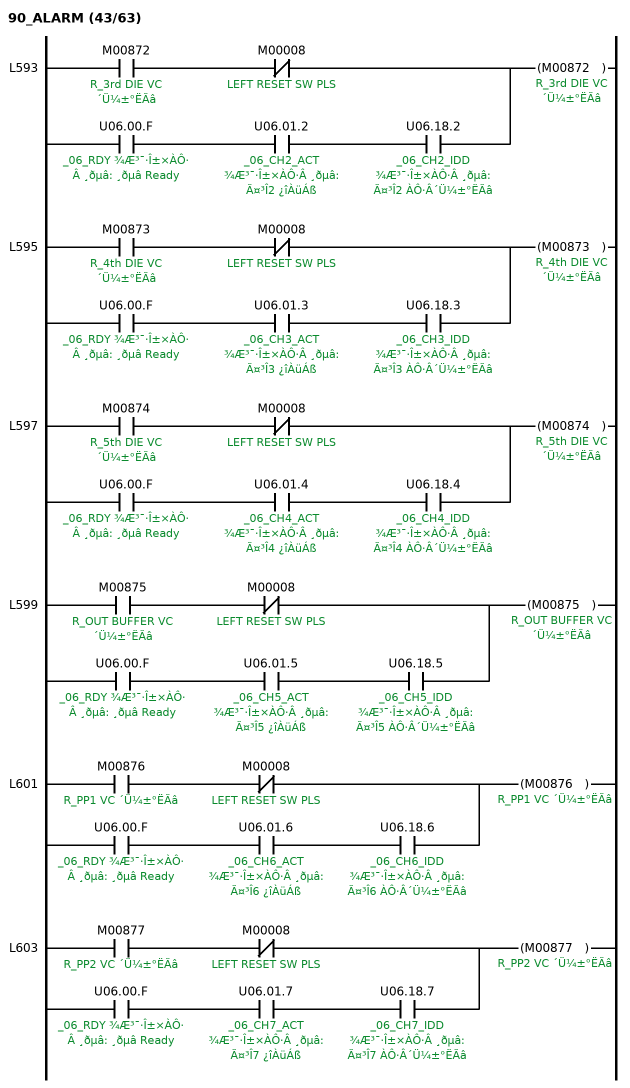
[picture p408: 90_ALARM rungs L593-L603]
; L593
LOAD      M00872	// R_3rd DIE VC ´Ü¼±°ËÃâ
AND NOT   M00008	// LEFT RESET SW PLS
LOAD      U06.00.F	// _06_RDY ¾Æ³¯·Î±×ÀÔ·Â ¸ðµâ: ¸ðµâ Ready
AND       U06.01.2	// _06_CH2_ACT ¾Æ³¯·Î±×ÀÔ·Â ¸ðµâ: Ã¤³Î2 ¿îÀüÁß
AND       U06.18.2	// _06_CH2_IDD ¾Æ³¯·Î±×ÀÔ·Â ¸ðµâ: Ã¤³Î2 ÀÔ·Â´Ü¼±°ËÃâ
OR LOAD
OUT       M00872	// R_3rd DIE VC ´Ü¼±°ËÃâ
; L595
LOAD      M00873	// R_4th DIE VC ´Ü¼±°ËÃâ
AND NOT   M00008	// LEFT RESET SW PLS
LOAD      U06.00.F	// _06_RDY ¾Æ³¯·Î±×ÀÔ·Â ¸ðµâ: ¸ðµâ Ready
AND       U06.01.3	// _06_CH3_ACT ¾Æ³¯·Î±×ÀÔ·Â ¸ðµâ: Ã¤³Î3 ¿îÀüÁß
AND       U06.18.3	// _06_CH3_IDD ¾Æ³¯·Î±×ÀÔ·Â ¸ðµâ: Ã¤³Î3 ÀÔ·Â´Ü¼±°ËÃâ
OR LOAD
OUT       M00873	// R_4th DIE VC ´Ü¼±°ËÃâ
; L597
LOAD      M00874	// R_5th DIE VC ´Ü¼±°ËÃâ
AND NOT   M00008	// LEFT RESET SW PLS
LOAD      U06.00.F	// _06_RDY ¾Æ³¯·Î±×ÀÔ·Â ¸ðµâ: ¸ðµâ Ready
AND       U06.01.4	// _06_CH4_ACT ¾Æ³¯·Î±×ÀÔ·Â ¸ðµâ: Ã¤³Î4 ¿îÀüÁß
AND       U06.18.4	// _06_CH4_IDD ¾Æ³¯·Î±×ÀÔ·Â ¸ðµâ: Ã¤³Î4 ÀÔ·Â´Ü¼±°ËÃâ
OR LOAD
OUT       M00874	// R_5th DIE VC ´Ü¼±°ËÃâ
; L599
LOAD      M00875	// R_OUT BUFFER VC ´Ü¼±°ËÃâ
AND NOT   M00008	// LEFT RESET SW PLS
LOAD      U06.00.F	// _06_RDY ¾Æ³¯·Î±×ÀÔ·Â ¸ðµâ: ¸ðµâ Ready
AND       U06.01.5	// _06_CH5_ACT ¾Æ³¯·Î±×ÀÔ·Â ¸ðµâ: Ã¤³Î5 ¿îÀüÁß
AND       U06.18.5	// _06_CH5_IDD ¾Æ³¯·Î±×ÀÔ·Â ¸ðµâ: Ã¤³Î5 ÀÔ·Â´Ü¼±°ËÃâ
OR LOAD
OUT       M00875	// R_OUT BUFFER VC ´Ü¼±°ËÃâ
; L601
LOAD      M00876	// R_PP1 VC ´Ü¼±°ËÃâ
AND NOT   M00008	// LEFT RESET SW PLS
LOAD      U06.00.F	// _06_RDY ¾Æ³¯·Î±×ÀÔ·Â ¸ðµâ: ¸ðµâ Ready
AND       U06.01.6	// _06_CH6_ACT ¾Æ³¯·Î±×ÀÔ·Â ¸ðµâ: Ã¤³Î6 ¿îÀüÁß
AND       U06.18.6	// _06_CH6_IDD ¾Æ³¯·Î±×ÀÔ·Â ¸ðµâ: Ã¤³Î6 ÀÔ·Â´Ü¼±°ËÃâ
OR LOAD
OUT       M00876	// R_PP1 VC ´Ü¼±°ËÃâ
; L603
LOAD      M00877	// R_PP2 VC ´Ü¼±°ËÃâ
AND NOT   M00008	// LEFT RESET SW PLS
LOAD      U06.00.F	// _06_RDY ¾Æ³¯·Î±×ÀÔ·Â ¸ðµâ: ¸ðµâ Ready
AND       U06.01.7	// _06_CH7_ACT ¾Æ³¯·Î±×ÀÔ·Â ¸ðµâ: Ã¤³Î7 ¿îÀüÁß
AND       U06.18.7	// _06_CH7_IDD ¾Æ³¯·Î±×ÀÔ·Â ¸ðµâ: Ã¤³Î7 ÀÔ·Â´Ü¼±°ËÃâ
OR LOAD
OUT       M00877	// R_PP2 VC ´Ü¼±°ËÃâ

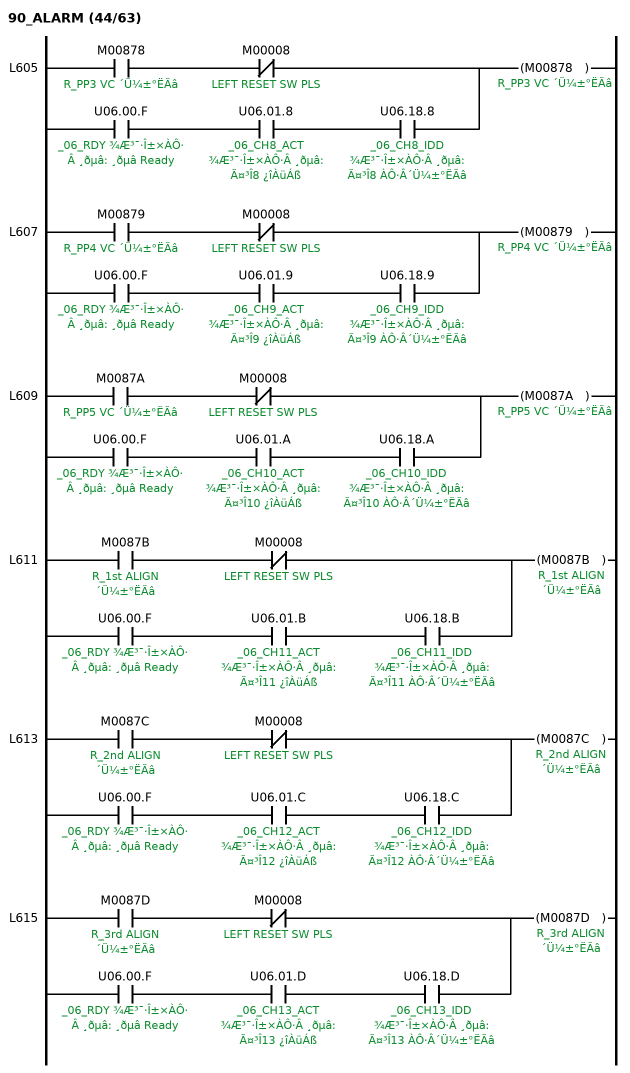
; L605
LOAD      M00878	// R_PP3 VC ´Ü¼±°ËÃâ
AND NOT   M00008	// LEFT RESET SW PLS
LOAD      U06.00.F	// _06_RDY ¾Æ³¯·Î±×ÀÔ·Â ¸ðµâ: ¸ðµâ Ready
AND       U06.01.8	// _06_CH8_ACT ¾Æ³¯·Î±×ÀÔ·Â ¸ðµâ: Ã¤³Î8 ¿îÀüÁß
AND       U06.18.8	// _06_CH8_IDD ¾Æ³¯·Î±×ÀÔ·Â ¸ðµâ: Ã¤³Î8 ÀÔ·Â´Ü¼±°ËÃâ
OR LOAD
OUT       M00878	// R_PP3 VC ´Ü¼±°ËÃâ
; L607
LOAD      M00879	// R_PP4 VC ´Ü¼±°ËÃâ
AND NOT   M00008	// LEFT RESET SW PLS
LOAD      U06.00.F	// _06_RDY ¾Æ³¯·Î±×ÀÔ·Â ¸ðµâ: ¸ðµâ Ready
AND       U06.01.9	// _06_CH9_ACT ¾Æ³¯·Î±×ÀÔ·Â ¸ðµâ: Ã¤³Î9 ¿îÀüÁß
AND       U06.18.9	// _06_CH9_IDD ¾Æ³¯·Î±×ÀÔ·Â ¸ðµâ: Ã¤³Î9 ÀÔ·Â´Ü¼±°ËÃâ
OR LOAD
OUT       M00879	// R_PP4 VC ´Ü¼±°ËÃâ
; L609
LOAD      M0087A	// R_PP5 VC ´Ü¼±°ËÃâ
AND NOT   M00008	// LEFT RESET SW PLS
LOAD      U06.00.F	// _06_RDY ¾Æ³¯·Î±×ÀÔ·Â ¸ðµâ: ¸ðµâ Ready
AND       U06.01.A	// _06_CH10_ACT ¾Æ³¯·Î±×ÀÔ·Â ¸ðµâ: Ã¤³Î10 ¿îÀüÁß
AND       U06.18.A	// _06_CH10_IDD ¾Æ³¯·Î±×ÀÔ·Â ¸ðµâ: Ã¤³Î10 ÀÔ·Â´Ü¼±°ËÃâ
OR LOAD
OUT       M0087A	// R_PP5 VC ´Ü¼±°ËÃâ
; L611
LOAD      M0087B	// R_1st ALIGN ´Ü¼±°ËÃâ
AND NOT   M00008	// LEFT RESET SW PLS
LOAD      U06.00.F	// _06_RDY ¾Æ³¯·Î±×ÀÔ·Â ¸ðµâ: ¸ðµâ Ready
AND       U06.01.B	// _06_CH11_ACT ¾Æ³¯·Î±×ÀÔ·Â ¸ðµâ: Ã¤³Î11 ¿îÀüÁß
AND       U06.18.B	// _06_CH11_IDD ¾Æ³¯·Î±×ÀÔ·Â ¸ðµâ: Ã¤³Î11 ÀÔ·Â´Ü¼±°ËÃâ
OR LOAD
OUT       M0087B	// R_1st ALIGN ´Ü¼±°ËÃâ
; L613
LOAD      M0087C	// R_2nd ALIGN ´Ü¼±°ËÃâ
AND NOT   M00008	// LEFT RESET SW PLS
LOAD      U06.00.F	// _06_RDY ¾Æ³¯·Î±×ÀÔ·Â ¸ðµâ: ¸ðµâ Ready
AND       U06.01.C	// _06_CH12_ACT ¾Æ³¯·Î±×ÀÔ·Â ¸ðµâ: Ã¤³Î12 ¿îÀüÁß
AND       U06.18.C	// _06_CH12_IDD ¾Æ³¯·Î±×ÀÔ·Â ¸ðµâ: Ã¤³Î12 ÀÔ·Â´Ü¼±°ËÃâ
OR LOAD
OUT       M0087C	// R_2nd ALIGN ´Ü¼±°ËÃâ
; L615
LOAD      M0087D	// R_3rd ALIGN ´Ü¼±°ËÃâ
AND NOT   M00008	// LEFT RESET SW PLS
LOAD      U06.00.F	// _06_RDY ¾Æ³¯·Î±×ÀÔ·Â ¸ðµâ: ¸ðµâ Ready
AND       U06.01.D	// _06_CH13_ACT ¾Æ³¯·Î±×ÀÔ·Â ¸ðµâ: Ã¤³Î13 ¿îÀüÁß
AND       U06.18.D	// _06_CH13_IDD ¾Æ³¯·Î±×ÀÔ·Â ¸ðµâ: Ã¤³Î13 ÀÔ·Â´Ü¼±°ËÃâ
OR LOAD
OUT       M0087D	// R_3rd ALIGN ´Ü¼±°ËÃâ

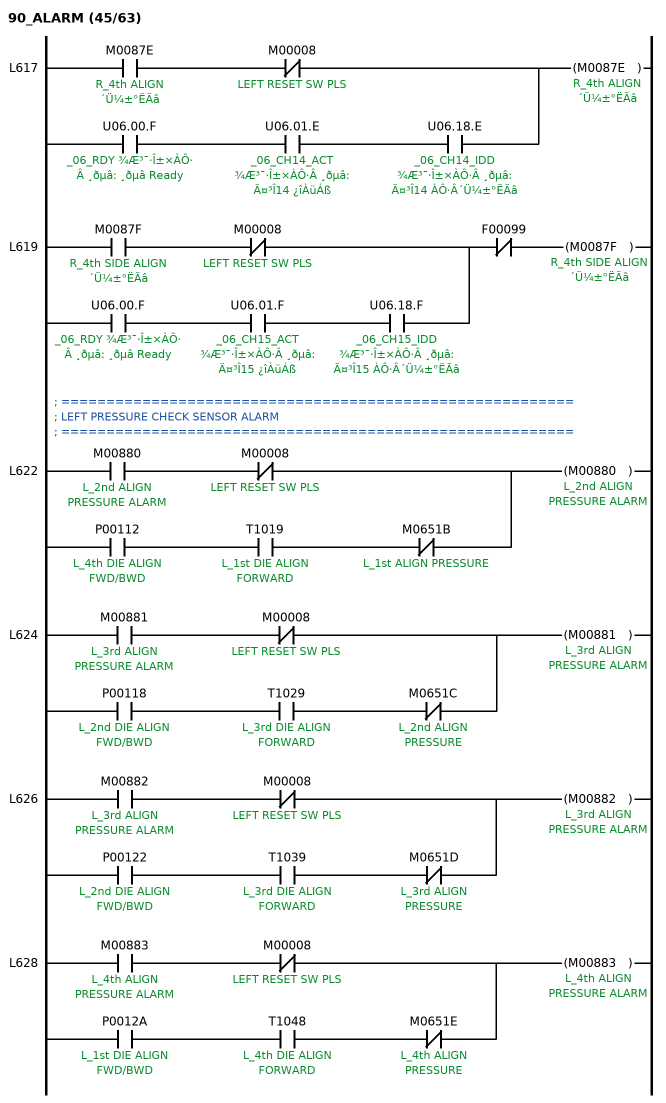
; L617
LOAD      M0087E	// R_4th ALIGN ´Ü¼±°ËÃâ
AND NOT   M00008	// LEFT RESET SW PLS
LOAD      U06.00.F	// _06_RDY ¾Æ³¯·Î±×ÀÔ·Â ¸ðµâ: ¸ðµâ Ready
AND       U06.01.E	// _06_CH14_ACT ¾Æ³¯·Î±×ÀÔ·Â ¸ðµâ: Ã¤³Î14 ¿îÀüÁß
AND       U06.18.E	// _06_CH14_IDD ¾Æ³¯·Î±×ÀÔ·Â ¸ðµâ: Ã¤³Î14 ÀÔ·Â´Ü¼±°ËÃâ
OR LOAD
OUT       M0087E	// R_4th ALIGN ´Ü¼±°ËÃâ
; L619
LOAD      M0087F	// R_4th SIDE ALIGN ´Ü¼±°ËÃâ
AND NOT   M00008	// LEFT RESET SW PLS
LOAD      U06.00.F	// _06_RDY ¾Æ³¯·Î±×ÀÔ·Â ¸ðµâ: ¸ðµâ Ready
AND       U06.01.F	// _06_CH15_ACT ¾Æ³¯·Î±×ÀÔ·Â ¸ðµâ: Ã¤³Î15 ¿îÀüÁß
AND       U06.18.F	// _06_CH15_IDD ¾Æ³¯·Î±×ÀÔ·Â ¸ðµâ: Ã¤³Î15 ÀÔ·Â´Ü¼±°ËÃâ
OR LOAD
AND NOT   F00099
OUT       M0087F	// R_4th SIDE ALIGN ´Ü¼±°ËÃâ
// =========================================================
// 
//        LEFT PRESSURE CHECK SENSOR ALARM
// 
// =========================================================
; L622
LOAD      M00880	// L_2nd ALIGN PRESSURE ALARM
AND NOT   M00008	// LEFT RESET SW PLS
LOAD      P00112	// L_4th DIE ALIGN FWD/BWD
AND       T1019	// L_1st DIE ALIGN FORWARD
AND NOT   M0651B	// L_1st ALIGN PRESSURE
OR LOAD
OUT       M00880	// L_2nd ALIGN PRESSURE ALARM
; L624
LOAD      M00881	// L_3rd ALIGN PRESSURE ALARM
AND NOT   M00008	// LEFT RESET SW PLS
LOAD      P00118	// L_2nd DIE ALIGN FWD/BWD
AND       T1029	// L_3rd DIE ALIGN FORWARD
AND NOT   M0651C	// L_2nd ALIGN PRESSURE
OR LOAD
OUT       M00881	// L_3rd ALIGN PRESSURE ALARM
; L626
LOAD      M00882	// L_3rd ALIGN PRESSURE ALARM
AND NOT   M00008	// LEFT RESET SW PLS
LOAD      P00122	// L_2nd DIE ALIGN FWD/BWD
AND       T1039	// L_3rd DIE ALIGN FORWARD
AND NOT   M0651D	// L_3rd ALIGN PRESSURE
OR LOAD
OUT       M00882	// L_3rd ALIGN PRESSURE ALARM
; L628
LOAD      M00883	// L_4th ALIGN PRESSURE ALARM
AND NOT   M00008	// LEFT RESET SW PLS
LOAD      P0012A	// L_1st DIE ALIGN FWD/BWD
AND       T1048	// L_4th DIE ALIGN FORWARD
AND NOT   M0651E	// L_4th ALIGN PRESSURE
OR LOAD
OUT       M00883	// L_4th ALIGN PRESSURE ALARM

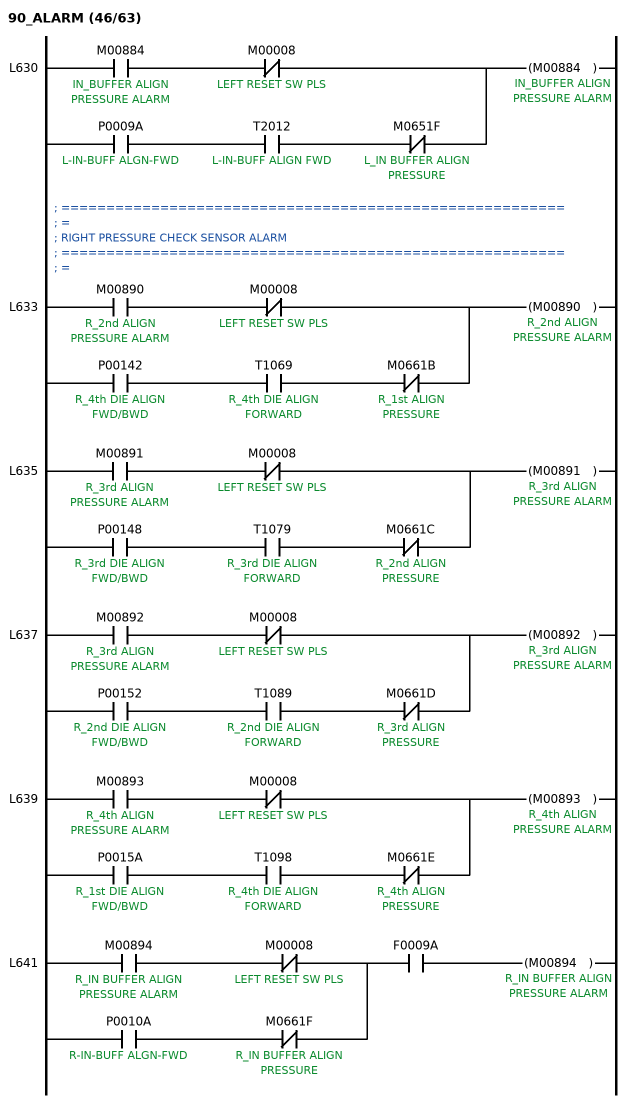
; L630
LOAD      M00884	// IN_BUFFER ALIGN PRESSURE ALARM
AND NOT   M00008	// LEFT RESET SW PLS
LOAD      P0009A	// L-IN-BUFF ALGN-FWD
AND       T2012	// L-IN-BUFF ALIGN FWD
AND NOT   M0651F	// L_IN BUFFER ALIGN PRESSURE
OR LOAD
OUT       M00884	// IN_BUFFER ALIGN PRESSURE ALARM
// =========================================================
// 
//        RIGHT PRESSURE CHECK SENSOR ALARM
// 
// =========================================================
; L633
LOAD      M00890	// R_2nd ALIGN PRESSURE ALARM
AND NOT   M00008	// LEFT RESET SW PLS
LOAD      P00142	// R_4th DIE ALIGN FWD/BWD
AND       T1069	// R_4th DIE ALIGN FORWARD
AND NOT   M0661B	// R_1st ALIGN PRESSURE
OR LOAD
OUT       M00890	// R_2nd ALIGN PRESSURE ALARM
; L635
LOAD      M00891	// R_3rd ALIGN PRESSURE ALARM
AND NOT   M00008	// LEFT RESET SW PLS
LOAD      P00148	// R_3rd DIE ALIGN FWD/BWD
AND       T1079	// R_3rd DIE ALIGN FORWARD
AND NOT   M0661C	// R_2nd ALIGN PRESSURE
OR LOAD
OUT       M00891	// R_3rd ALIGN PRESSURE ALARM
; L637
LOAD      M00892	// R_3rd ALIGN PRESSURE ALARM
AND NOT   M00008	// LEFT RESET SW PLS
LOAD      P00152	// R_2nd DIE ALIGN FWD/BWD
AND       T1089	// R_2nd DIE ALIGN FORWARD
AND NOT   M0661D	// R_3rd ALIGN PRESSURE
OR LOAD
OUT       M00892	// R_3rd ALIGN PRESSURE ALARM
; L639
LOAD      M00893	// R_4th ALIGN PRESSURE ALARM
AND NOT   M00008	// LEFT RESET SW PLS
LOAD      P0015A	// R_1st DIE ALIGN FWD/BWD
AND       T1098	// R_4th DIE ALIGN FORWARD
AND NOT   M0661E	// R_4th ALIGN PRESSURE
OR LOAD
OUT       M00893	// R_4th ALIGN PRESSURE ALARM
; L641
LOAD      M00894	// R_IN BUFFER ALIGN PRESSURE ALARM
AND NOT   M00008	// LEFT RESET SW PLS
LOAD      P0010A	// R-IN-BUFF ALGN-FWD
AND NOT   M0661F	// R_IN BUFFER ALIGN PRESSURE
OR LOAD
AND       F0009A
OUT       M00894	// R_IN BUFFER ALIGN PRESSURE ALARM

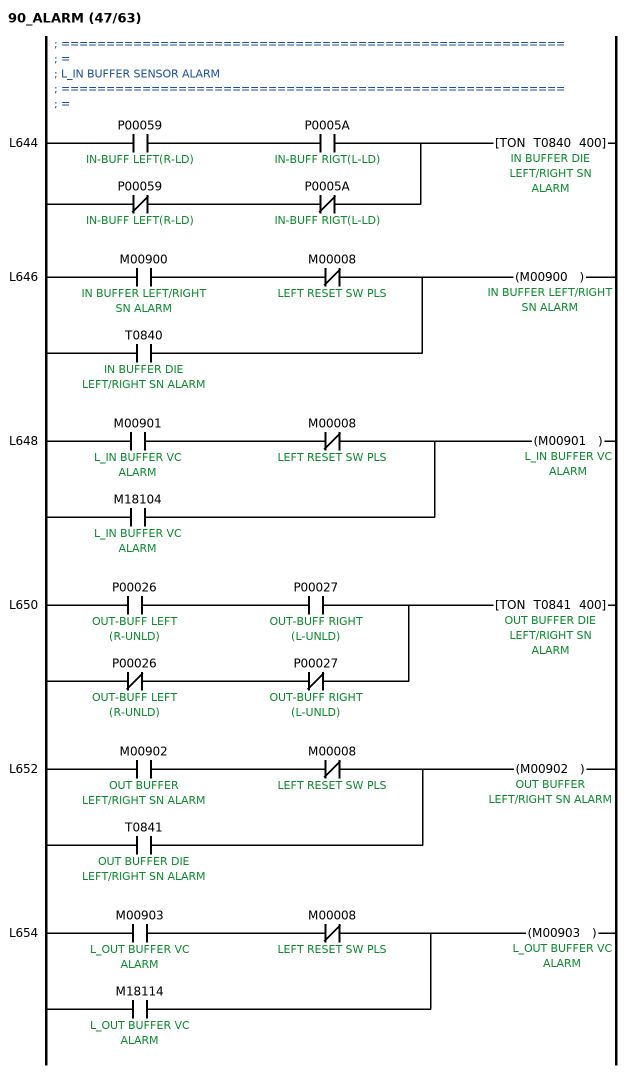
// =========================================================
// 
//        L_IN BUFFER SENSOR ALARM
// 
// =========================================================
; L644
LOAD      P00059	// IN-BUFF LEFT(R-LD)
AND       P0005A	// IN-BUFF RIGT(L-LD)
LOAD NOT  P00059	// IN-BUFF LEFT(R-LD)
AND NOT   P0005A	// IN-BUFF RIGT(L-LD)
OR LOAD
TON       T0840 400	// IN BUFFER DIE LEFT/RIGHT SN ALARM
; L646
LOAD      M00900	// IN BUFFER LEFT/RIGHT SN ALARM
AND NOT   M00008	// LEFT RESET SW PLS
OR        T0840	// IN BUFFER DIE LEFT/RIGHT SN ALARM
OUT       M00900	// IN BUFFER LEFT/RIGHT SN ALARM
; L648
LOAD      M00901	// L_IN BUFFER VC ALARM
AND NOT   M00008	// LEFT RESET SW PLS
OR        M18104	// L_IN BUFFER VC ALARM
OUT       M00901	// L_IN BUFFER VC ALARM
; L650
LOAD      P00026	// OUT-BUFF LEFT (R-UNLD)
AND       P00027	// OUT-BUFF RIGHT (L-UNLD)
LOAD NOT  P00026	// OUT-BUFF LEFT (R-UNLD)
AND NOT   P00027	// OUT-BUFF RIGHT (L-UNLD)
OR LOAD
TON       T0841 400	// OUT BUFFER DIE LEFT/RIGHT SN ALARM
; L652
LOAD      M00902	// OUT BUFFER LEFT/RIGHT SN ALARM
AND NOT   M00008	// LEFT RESET SW PLS
OR        T0841	// OUT BUFFER DIE LEFT/RIGHT SN ALARM
OUT       M00902	// OUT BUFFER LEFT/RIGHT SN ALARM
; L654
LOAD      M00903	// L_OUT BUFFER VC ALARM
AND NOT   M00008	// LEFT RESET SW PLS
OR        M18114	// L_OUT BUFFER VC ALARM
OUT       M00903	// L_OUT BUFFER VC ALARM

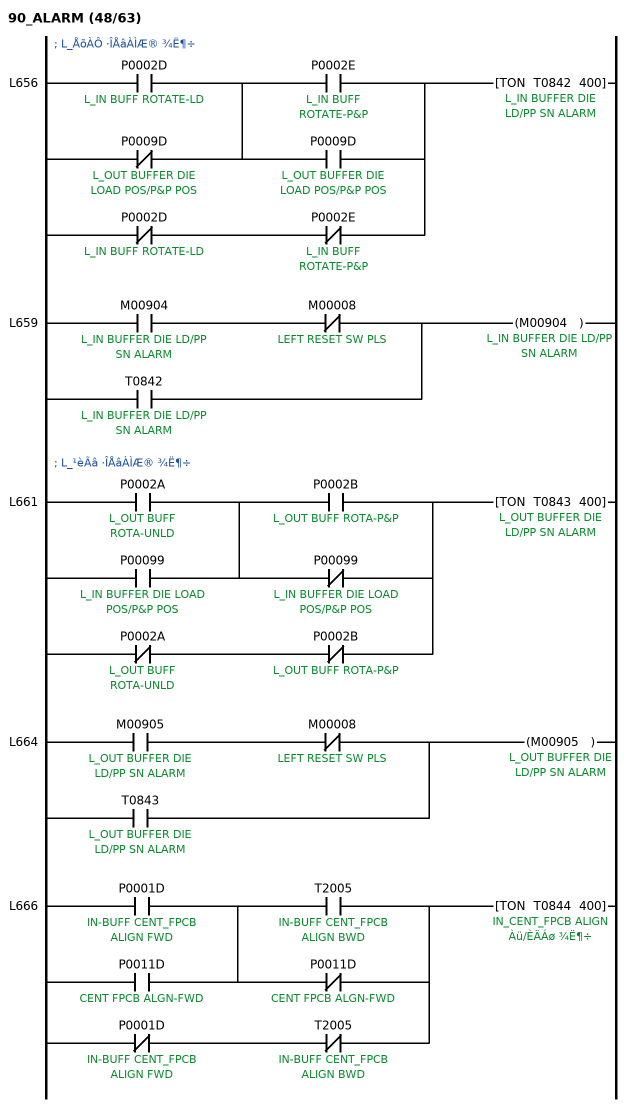
; L656
LOAD      P0002D	// L_IN BUFF ROTATE-LD
OR NOT    P0009D	// L_OUT BUFFER DIE LOAD POS/P&P POS
LOAD      P0002E	// L_IN BUFF ROTATE-P&P
OR        P0009D	// L_OUT BUFFER DIE LOAD POS/P&P POS
AND LOAD
LOAD NOT  P0002D	// L_IN BUFF ROTATE-LD
AND NOT   P0002E	// L_IN BUFF ROTATE-P&P
OR LOAD
TON       T0842 400	// L_IN BUFFER DIE LD/PP SN ALARM
// output comment: L_ÅõÀÔ ·ÎÅâÀÌÆ® ¾Ë¶÷
; L659
LOAD      M00904	// L_IN BUFFER DIE LD/PP SN ALARM
AND NOT   M00008	// LEFT RESET SW PLS
OR        T0842	// L_IN BUFFER DIE LD/PP SN ALARM
OUT       M00904	// L_IN BUFFER DIE LD/PP SN ALARM
; L661
LOAD      P0002A	// L_OUT BUFF ROTA-UNLD
OR        P00099	// L_IN BUFFER DIE LOAD POS/P&P POS
LOAD      P0002B	// L_OUT BUFF ROTA-P&P
OR NOT    P00099	// L_IN BUFFER DIE LOAD POS/P&P POS
AND LOAD
LOAD NOT  P0002A	// L_OUT BUFF ROTA-UNLD
AND NOT   P0002B	// L_OUT BUFF ROTA-P&P
OR LOAD
TON       T0843 400	// L_OUT BUFFER DIE LD/PP SN ALARM
// output comment: L_¹èÃâ ·ÎÅâÀÌÆ® ¾Ë¶÷
; L664
LOAD      M00905	// L_OUT BUFFER DIE LD/PP SN ALARM
AND NOT   M00008	// LEFT RESET SW PLS
OR        T0843	// L_OUT BUFFER DIE LD/PP SN ALARM
OUT       M00905	// L_OUT BUFFER DIE LD/PP SN ALARM
; L666
LOAD      P0001D	// IN-BUFF CENT_FPCB ALIGN FWD
OR        P0011D	// CENT FPCB ALGN-FWD
LOAD      T2005	// IN-BUFF CENT_FPCB ALIGN BWD
OR NOT    P0011D	// CENT FPCB ALGN-FWD
AND LOAD
LOAD NOT  P0001D	// IN-BUFF CENT_FPCB ALIGN FWD
AND NOT   T2005	// IN-BUFF CENT_FPCB ALIGN BWD
OR LOAD
TON       T0844 400	// IN_CENT_FPCB ALIGN Àü/ÈÄÁø ¾Ë¶÷

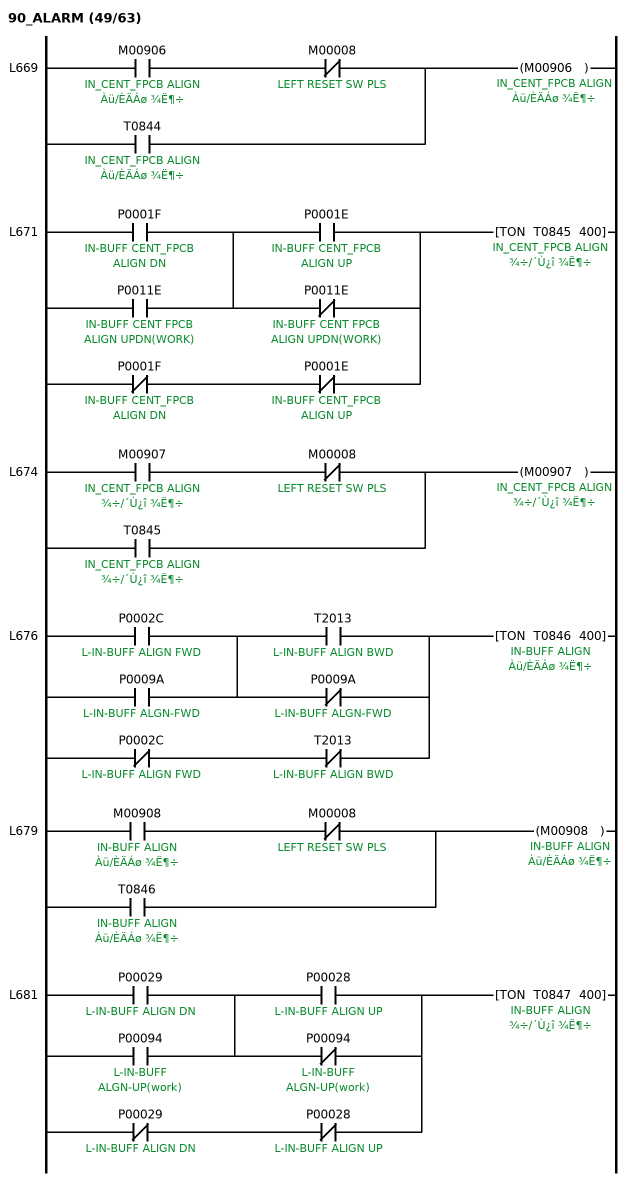
; L669
LOAD      M00906	// IN_CENT_FPCB ALIGN Àü/ÈÄÁø ¾Ë¶÷
AND NOT   M00008	// LEFT RESET SW PLS
OR        T0844	// IN_CENT_FPCB ALIGN Àü/ÈÄÁø ¾Ë¶÷
OUT       M00906	// IN_CENT_FPCB ALIGN Àü/ÈÄÁø ¾Ë¶÷
; L671
LOAD      P0001F	// IN-BUFF CENT_FPCB ALIGN DN
OR        P0011E	// IN-BUFF CENT FPCB ALIGN UPDN(WORK)
LOAD      P0001E	// IN-BUFF CENT_FPCB ALIGN UP
OR NOT    P0011E	// IN-BUFF CENT FPCB ALIGN UPDN(WORK)
AND LOAD
LOAD NOT  P0001F	// IN-BUFF CENT_FPCB ALIGN DN
AND NOT   P0001E	// IN-BUFF CENT_FPCB ALIGN UP
OR LOAD
TON       T0845 400	// IN_CENT_FPCB ALIGN ¾÷/´Ù¿î ¾Ë¶÷
; L674
LOAD      M00907	// IN_CENT_FPCB ALIGN ¾÷/´Ù¿î ¾Ë¶÷
AND NOT   M00008	// LEFT RESET SW PLS
OR        T0845	// IN_CENT_FPCB ALIGN ¾÷/´Ù¿î ¾Ë¶÷
OUT       M00907	// IN_CENT_FPCB ALIGN ¾÷/´Ù¿î ¾Ë¶÷
; L676
LOAD      P0002C	// L-IN-BUFF ALIGN FWD
OR        P0009A	// L-IN-BUFF ALGN-FWD
LOAD      T2013	// L-IN-BUFF ALIGN BWD
OR NOT    P0009A	// L-IN-BUFF ALGN-FWD
AND LOAD
LOAD NOT  P0002C	// L-IN-BUFF ALIGN FWD
AND NOT   T2013	// L-IN-BUFF ALIGN BWD
OR LOAD
TON       T0846 400	// IN-BUFF ALIGN Àü/ÈÄÁø ¾Ë¶÷
; L679
LOAD      M00908	// IN-BUFF ALIGN Àü/ÈÄÁø ¾Ë¶÷
AND NOT   M00008	// LEFT RESET SW PLS
OR        T0846	// IN-BUFF ALIGN Àü/ÈÄÁø ¾Ë¶÷
OUT       M00908	// IN-BUFF ALIGN Àü/ÈÄÁø ¾Ë¶÷
; L681
LOAD      P00029	// L-IN-BUFF ALIGN DN
OR        P00094	// L-IN-BUFF ALGN-UP(work)
LOAD      P00028	// L-IN-BUFF ALIGN UP
OR NOT    P00094	// L-IN-BUFF ALGN-UP(work)
AND LOAD
LOAD NOT  P00029	// L-IN-BUFF ALIGN DN
AND NOT   P00028	// L-IN-BUFF ALIGN UP
OR LOAD
TON       T0847 400	// IN-BUFF ALIGN ¾÷/´Ù¿î ¾Ë¶÷

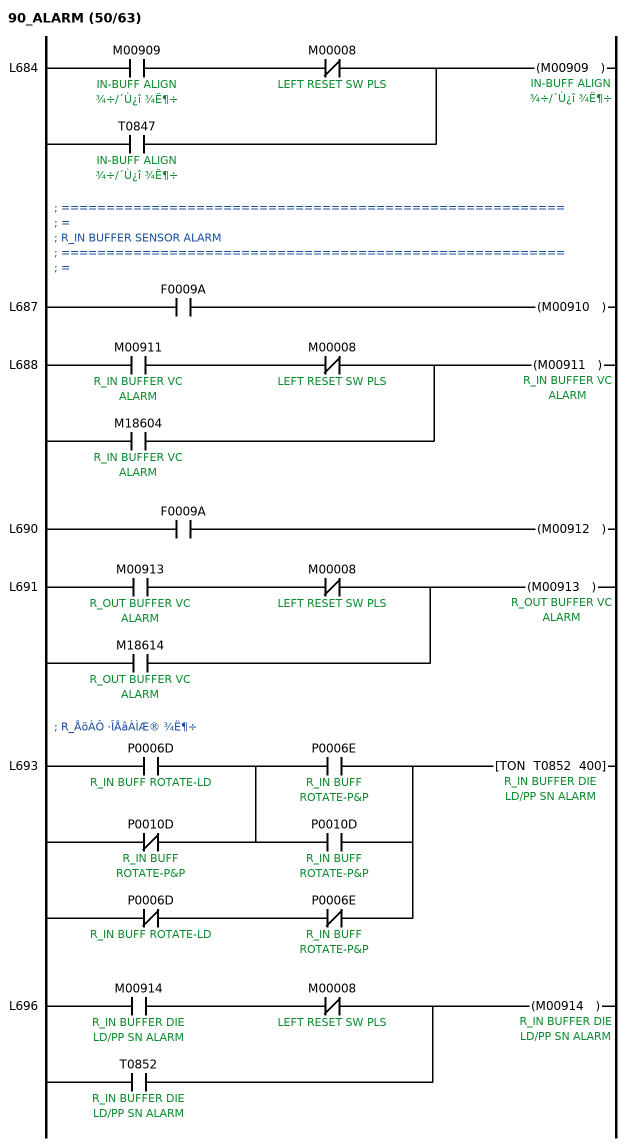
; L684
LOAD      M00909	// IN-BUFF ALIGN ¾÷/´Ù¿î ¾Ë¶÷
AND NOT   M00008	// LEFT RESET SW PLS
OR        T0847	// IN-BUFF ALIGN ¾÷/´Ù¿î ¾Ë¶÷
OUT       M00909	// IN-BUFF ALIGN ¾÷/´Ù¿î ¾Ë¶÷
// =========================================================
// 
//        R_IN BUFFER SENSOR ALARM
// 
// =========================================================
; L687
LOAD      F0009A
OUT       M00910
; L688
LOAD      M00911	// R_IN BUFFER VC ALARM
AND NOT   M00008	// LEFT RESET SW PLS
OR        M18604	// R_IN BUFFER VC ALARM
OUT       M00911	// R_IN BUFFER VC ALARM
; L690
LOAD      F0009A
OUT       M00912
; L691
LOAD      M00913	// R_OUT BUFFER VC ALARM
AND NOT   M00008	// LEFT RESET SW PLS
OR        M18614	// R_OUT BUFFER VC ALARM
OUT       M00913	// R_OUT BUFFER VC ALARM
; L693
LOAD      P0006D	// R_IN BUFF ROTATE-LD
OR NOT    P0010D	// R_IN BUFF ROTATE-P&P
LOAD      P0006E	// R_IN BUFF ROTATE-P&P
OR        P0010D	// R_IN BUFF ROTATE-P&P
AND LOAD
LOAD NOT  P0006D	// R_IN BUFF ROTATE-LD
AND NOT   P0006E	// R_IN BUFF ROTATE-P&P
OR LOAD
TON       T0852 400	// R_IN BUFFER DIE LD/PP SN ALARM
// output comment: R_ÅõÀÔ ·ÎÅâÀÌÆ® ¾Ë¶÷
; L696
LOAD      M00914	// R_IN BUFFER DIE LD/PP SN ALARM
AND NOT   M00008	// LEFT RESET SW PLS
OR        T0852	// R_IN BUFFER DIE LD/PP SN ALARM
OUT       M00914	// R_IN BUFFER DIE LD/PP SN ALARM

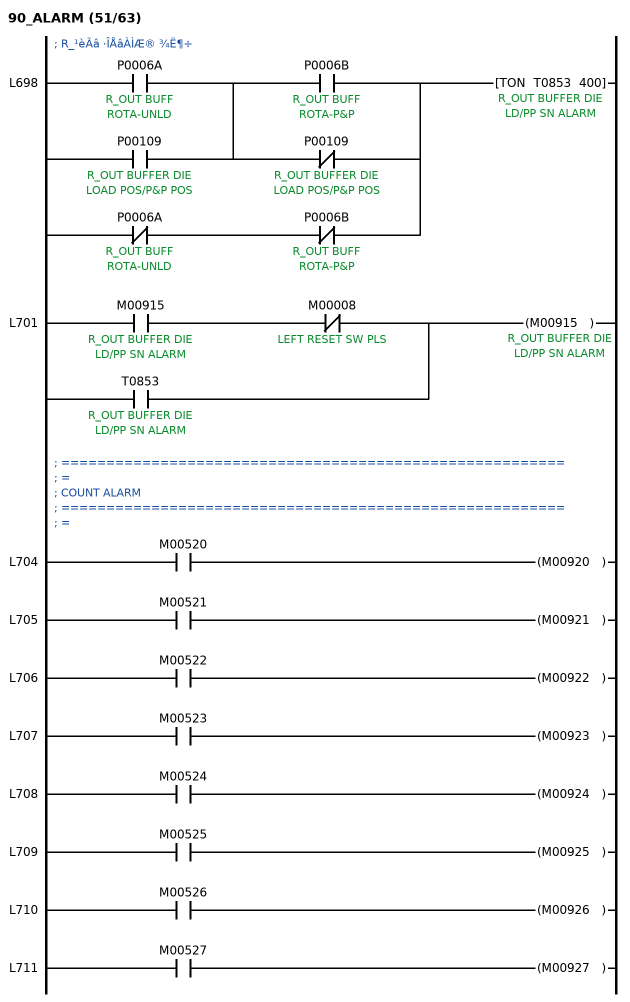
; L698
LOAD      P0006A	// R_OUT BUFF ROTA-UNLD
OR        P00109	// R_OUT BUFFER DIE LOAD POS/P&P POS
LOAD      P0006B	// R_OUT BUFF ROTA-P&P
OR NOT    P00109	// R_OUT BUFFER DIE LOAD POS/P&P POS
AND LOAD
LOAD NOT  P0006A	// R_OUT BUFF ROTA-UNLD
AND NOT   P0006B	// R_OUT BUFF ROTA-P&P
OR LOAD
TON       T0853 400	// R_OUT BUFFER DIE LD/PP SN ALARM
// output comment: R_¹èÃâ ·ÎÅâÀÌÆ® ¾Ë¶÷
; L701
LOAD      M00915	// R_OUT BUFFER DIE LD/PP SN ALARM
AND NOT   M00008	// LEFT RESET SW PLS
OR        T0853	// R_OUT BUFFER DIE LD/PP SN ALARM
OUT       M00915	// R_OUT BUFFER DIE LD/PP SN ALARM
// =========================================================
// 
//       COUNT ALARM
// 
// =========================================================
; L704
LOAD      M00520
OUT       M00920
; L705
LOAD      M00521
OUT       M00921
; L706
LOAD      M00522
OUT       M00922
; L707
LOAD      M00523
OUT       M00923
; L708
LOAD      M00524
OUT       M00924
; L709
LOAD      M00525
OUT       M00925
; L710
LOAD      M00526
OUT       M00926
; L711
LOAD      M00527
OUT       M00927

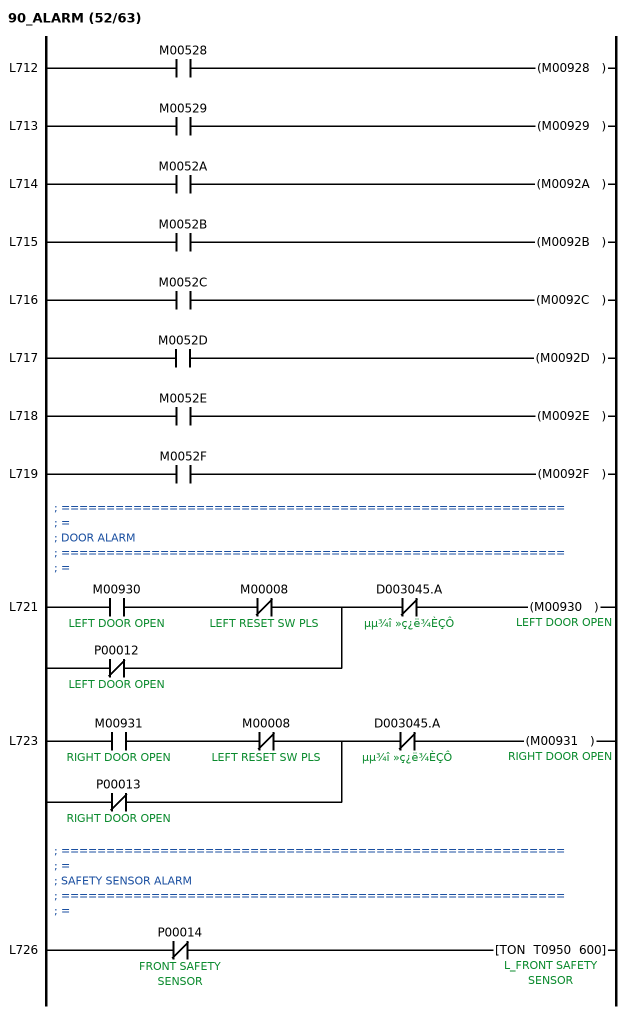
; L712
LOAD      M00528
OUT       M00928
; L713
LOAD      M00529
OUT       M00929
; L714
LOAD      M0052A
OUT       M0092A
; L715
LOAD      M0052B
OUT       M0092B
; L716
LOAD      M0052C
OUT       M0092C
; L717
LOAD      M0052D
OUT       M0092D
; L718
LOAD      M0052E
OUT       M0092E
; L719
LOAD      M0052F
OUT       M0092F
// =========================================================
// 
//       DOOR ALARM
// 
// =========================================================
; L721
LOAD      M00930	// LEFT DOOR OPEN
AND NOT   M00008	// LEFT RESET SW PLS
OR NOT    P00012	// LEFT DOOR OPEN
AND NOT   D003045.A	// µµ¾î »ç¿ë¾ÈÇÔ
OUT       M00930	// LEFT DOOR OPEN
; L723
LOAD      M00931	// RIGHT DOOR OPEN
AND NOT   M00008	// LEFT RESET SW PLS
OR NOT    P00013	// RIGHT DOOR OPEN
AND NOT   D003045.A	// µµ¾î »ç¿ë¾ÈÇÔ
OUT       M00931	// RIGHT DOOR OPEN
// =========================================================
// 
//       SAFETY SENSOR ALARM
// 
// =========================================================
; L726
LOAD NOT  P00014	// FRONT SAFETY SENSOR
TON       T0950 600	// L_FRONT SAFETY SENSOR

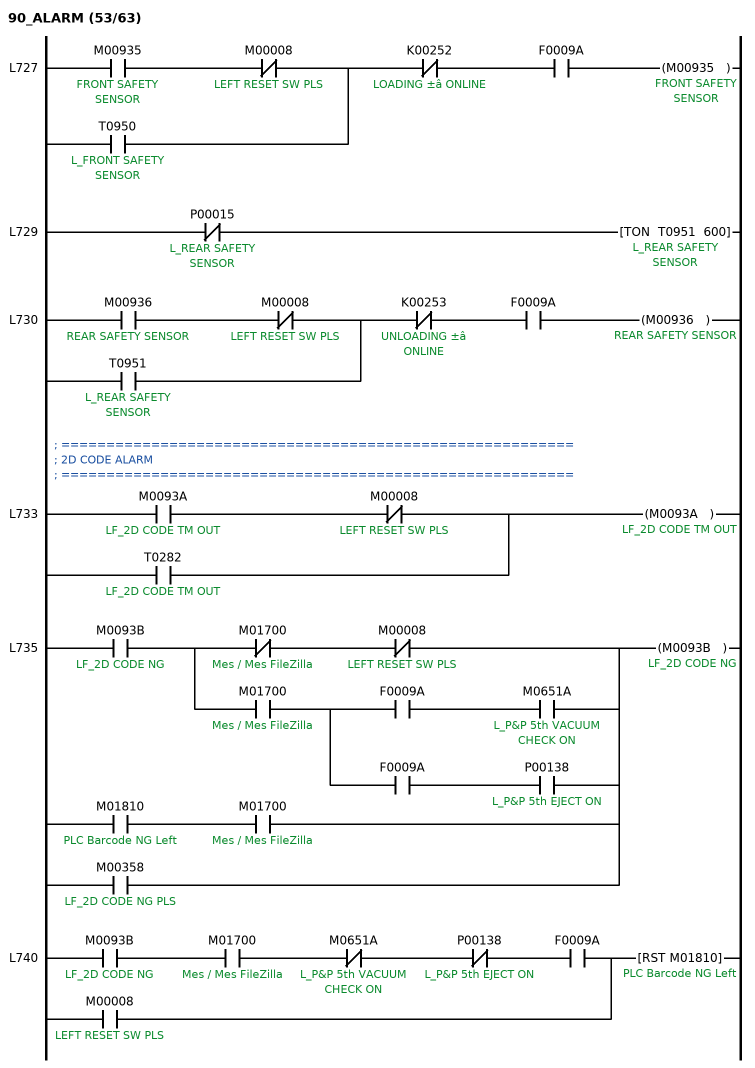
; L727
LOAD      M00935	// FRONT SAFETY SENSOR
AND NOT   M00008	// LEFT RESET SW PLS
OR        T0950	// L_FRONT SAFETY SENSOR
AND NOT   K00252	// LOADING ±â ONLINE
AND       F0009A
OUT       M00935	// FRONT SAFETY SENSOR
; L729
LOAD NOT  P00015	// L_REAR SAFETY SENSOR
TON       T0951 600	// L_REAR SAFETY SENSOR
; L730
LOAD      M00936	// REAR SAFETY SENSOR
AND NOT   M00008	// LEFT RESET SW PLS
OR        T0951	// L_REAR SAFETY SENSOR
AND NOT   K00253	// UNLOADING ±â ONLINE
AND       F0009A
OUT       M00936	// REAR SAFETY SENSOR
// =========================================================
// 
//       2D CODE ALARM
// 
// =========================================================
; L733
LOAD      M0093A	// LF_2D CODE TM OUT
AND NOT   M00008	// LEFT RESET SW PLS
OR        T0282	// LF_2D CODE TM OUT
OUT       M0093A	// LF_2D CODE TM OUT
; L735
LOAD      M0093B	// LF_2D CODE NG
LOAD NOT  M01700	// Mes / Mes FileZilla
AND NOT   M00008	// LEFT RESET SW PLS
LOAD      M01700	// Mes / Mes FileZilla
LOAD      F0009A
AND       M0651A	// L_P&P 5th VACUUM CHECK ON
LOAD      F0009A
AND       P00138	// L_P&P 5th EJECT ON
OR LOAD
AND LOAD
OR LOAD
AND LOAD
LOAD      M01810	// PLC Barcode NG Left
AND       M01700	// Mes / Mes FileZilla
OR LOAD
OR        M00358	// LF_2D CODE NG PLS
OUT       M0093B	// LF_2D CODE NG
; L740
LOAD      M0093B	// LF_2D CODE NG
AND       M01700	// Mes / Mes FileZilla
AND NOT   M0651A	// L_P&P 5th VACUUM CHECK ON
AND NOT   P00138	// L_P&P 5th EJECT ON
AND       F0009A
OR        M00008	// LEFT RESET SW PLS
RST       M01810	// PLC Barcode NG Left

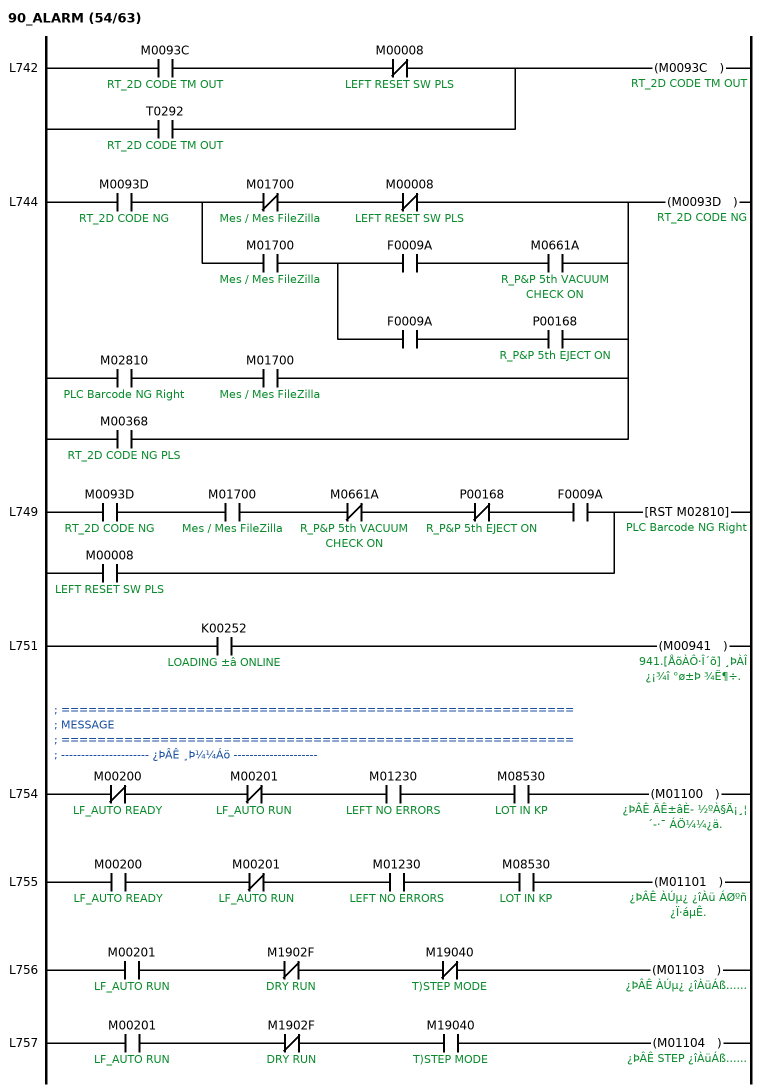
; L742
LOAD      M0093C	// RT_2D CODE TM OUT
AND NOT   M00008	// LEFT RESET SW PLS
OR        T0292	// RT_2D CODE TM OUT
OUT       M0093C	// RT_2D CODE TM OUT
; L744
LOAD      M0093D	// RT_2D CODE NG
LOAD NOT  M01700	// Mes / Mes FileZilla
AND NOT   M00008	// LEFT RESET SW PLS
LOAD      M01700	// Mes / Mes FileZilla
LOAD      F0009A
AND       M0661A	// R_P&P 5th VACUUM CHECK ON
LOAD      F0009A
AND       P00168	// R_P&P 5th EJECT ON
OR LOAD
AND LOAD
OR LOAD
AND LOAD
LOAD      M02810	// PLC Barcode NG Right
AND       M01700	// Mes / Mes FileZilla
OR LOAD
OR        M00368	// RT_2D CODE NG PLS
OUT       M0093D	// RT_2D CODE NG
; L749
LOAD      M0093D	// RT_2D CODE NG
AND       M01700	// Mes / Mes FileZilla
AND NOT   M0661A	// R_P&P 5th VACUUM CHECK ON
AND NOT   P00168	// R_P&P 5th EJECT ON
AND       F0009A
OR        M00008	// LEFT RESET SW PLS
RST       M02810	// PLC Barcode NG Right
; L751
LOAD      K00252	// LOADING ±â ONLINE
OUT       M00941	// 941.[ÅõÀÔ·Î´õ] ¸ÞÀÎ ¿¡¾î °ø±Þ ¾Ë¶÷.
// =========================================================
// 
//       MESSAGE
// 
// =========================================================
// ---------------------- ¿ÞÂÊ ¸Þ¼¼Áö ---------------------
; L754
LOAD NOT  M00200	// LF_AUTO READY
AND NOT   M00201	// LF_AUTO RUN
AND       M01230	// LEFT NO ERRORS
AND       M08530	// LOT IN KP
OUT       M01100	// ¿ÞÂÊ ÃÊ±âÈ­ ½ºÀ§Ä¡¸¦ ´­·¯ ÁÖ¼¼¿ä.
; L755
LOAD      M00200	// LF_AUTO READY
AND NOT   M00201	// LF_AUTO RUN
AND       M01230	// LEFT NO ERRORS
AND       M08530	// LOT IN KP
OUT       M01101	// ¿ÞÂÊ ÀÚµ¿ ¿îÀü ÁØºñ ¿Ï·áµÊ.
; L756
LOAD      M00201	// LF_AUTO RUN
AND NOT   M1902F	// DRY RUN
AND NOT   M19040	// T)STEP MODE
OUT       M01103	// ¿ÞÂÊ ÀÚµ¿ ¿îÀüÁß......
; L757
LOAD      M00201	// LF_AUTO RUN
AND NOT   M1902F	// DRY RUN
AND       M19040	// T)STEP MODE
OUT       M01104	// ¿ÞÂÊ STEP ¿îÀüÁß......

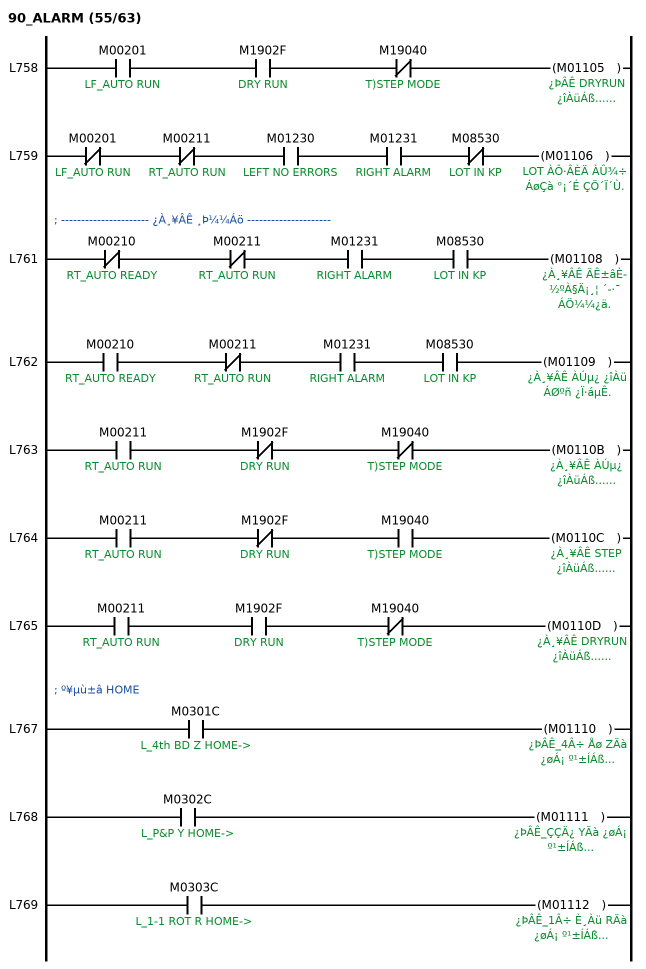
; L758
LOAD      M00201	// LF_AUTO RUN
AND       M1902F	// DRY RUN
AND NOT   M19040	// T)STEP MODE
OUT       M01105	// ¿ÞÂÊ DRYRUN ¿îÀüÁß......
; L759
LOAD NOT  M00201	// LF_AUTO RUN
AND NOT   M00211	// RT_AUTO RUN
AND       M01230	// LEFT NO ERRORS
AND       M01231	// RIGHT ALARM
AND NOT   M08530	// LOT IN KP
OUT       M01106	// LOT ÀÔ·ÂÈÄ ÀÛ¾÷ ÁøÇà °¡´É ÇÕ´Ï´Ù.
// ---------------------- ¿À¸¥ÂÊ ¸Þ¼¼Áö ---------------------
; L761
LOAD NOT  M00210	// RT_AUTO READY
AND NOT   M00211	// RT_AUTO RUN
AND       M01231	// RIGHT ALARM
AND       M08530	// LOT IN KP
OUT       M01108	// ¿À¸¥ÂÊ ÃÊ±âÈ­ ½ºÀ§Ä¡¸¦ ´­·¯ ÁÖ¼¼¿ä.
; L762
LOAD      M00210	// RT_AUTO READY
AND NOT   M00211	// RT_AUTO RUN
AND       M01231	// RIGHT ALARM
AND       M08530	// LOT IN KP
OUT       M01109	// ¿À¸¥ÂÊ ÀÚµ¿ ¿îÀü ÁØºñ ¿Ï·áµÊ.
; L763
LOAD      M00211	// RT_AUTO RUN
AND NOT   M1902F	// DRY RUN
AND NOT   M19040	// T)STEP MODE
OUT       M0110B	// ¿À¸¥ÂÊ ÀÚµ¿ ¿îÀüÁß......
; L764
LOAD      M00211	// RT_AUTO RUN
AND NOT   M1902F	// DRY RUN
AND       M19040	// T)STEP MODE
OUT       M0110C	// ¿À¸¥ÂÊ STEP ¿îÀüÁß......
; L765
LOAD      M00211	// RT_AUTO RUN
AND       M1902F	// DRY RUN
AND NOT   M19040	// T)STEP MODE
OUT       M0110D	// ¿À¸¥ÂÊ DRYRUN ¿îÀüÁß......
// º¥µù±â HOME
; L767
LOAD      M0301C	// L_4th BD Z HOME->
OUT       M01110	// ¿ÞÂÊ_4Â÷ Åø ZÃà ¿øÁ¡ º¹±ÍÁß...
; L768
LOAD      M0302C	// L_P&P Y HOME->
OUT       M01111	// ¿ÞÂÊ_ÇÇÄ¿ YÃà ¿øÁ¡ º¹±ÍÁß...
; L769
LOAD      M0303C	// L_1-1 ROT R HOME->
OUT       M01112	// ¿ÞÂÊ_1Â÷ È¸Àü RÃà ¿øÁ¡ º¹±ÍÁß...

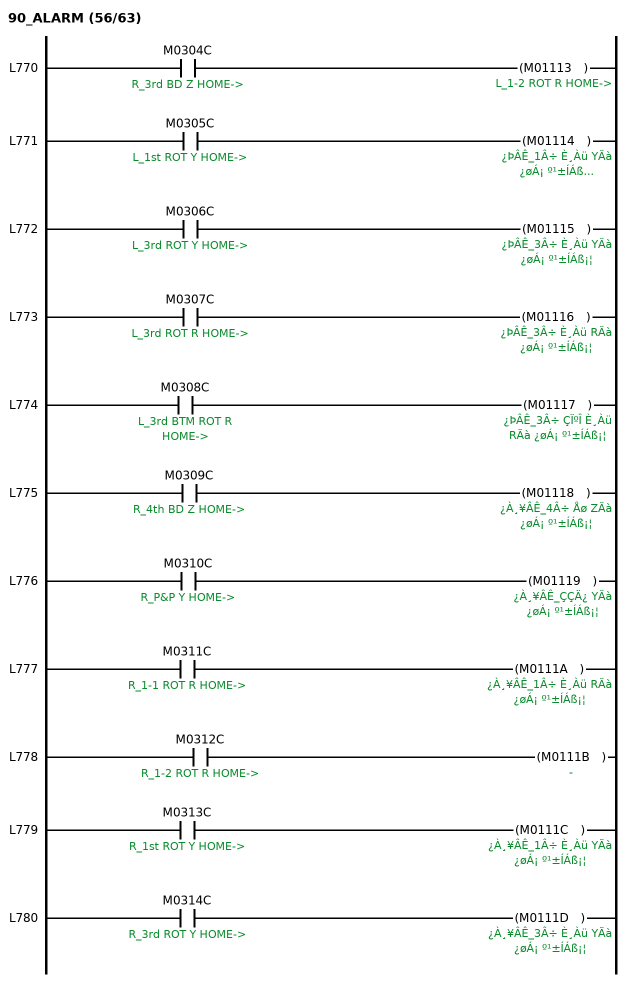
; L770
LOAD      M0304C	// R_3rd BD Z HOME->
OUT       M01113	// L_1-2 ROT R HOME->
; L771
LOAD      M0305C	// L_1st ROT Y HOME->
OUT       M01114	// ¿ÞÂÊ_1Â÷ È¸Àü YÃà ¿øÁ¡ º¹±ÍÁß...
; L772
LOAD      M0306C	// L_3rd ROT Y HOME->
OUT       M01115	// ¿ÞÂÊ_3Â÷ È¸Àü YÃà ¿øÁ¡ º¹±ÍÁß¡¦
; L773
LOAD      M0307C	// L_3rd ROT R HOME->
OUT       M01116	// ¿ÞÂÊ_3Â÷ È¸Àü RÃà ¿øÁ¡ º¹±ÍÁß¡¦
; L774
LOAD      M0308C	// L_3rd BTM ROT R HOME->
OUT       M01117	// ¿ÞÂÊ_3Â÷ ÇÏºÎ È¸Àü RÃà ¿øÁ¡ º¹±ÍÁß¡¦
; L775
LOAD      M0309C	// R_4th BD Z HOME->
OUT       M01118	// ¿À¸¥ÂÊ_4Â÷ Åø ZÃà ¿øÁ¡ º¹±ÍÁß¡¦
; L776
LOAD      M0310C	// R_P&P Y HOME->
OUT       M01119	// ¿À¸¥ÂÊ_ÇÇÄ¿ YÃà ¿øÁ¡ º¹±ÍÁß¡¦
; L777
LOAD      M0311C	// R_1-1 ROT R HOME->
OUT       M0111A	// ¿À¸¥ÂÊ_1Â÷ È¸Àü RÃà ¿øÁ¡ º¹±ÍÁß¡¦
; L778
LOAD      M0312C	// R_1-2 ROT R HOME->
OUT       M0111B	// -
; L779
LOAD      M0313C	// R_1st ROT Y HOME->
OUT       M0111C	// ¿À¸¥ÂÊ_1Â÷ È¸Àü YÃà ¿øÁ¡ º¹±ÍÁß¡¦
; L780
LOAD      M0314C	// R_3rd ROT Y HOME->
OUT       M0111D	// ¿À¸¥ÂÊ_3Â÷ È¸Àü YÃà ¿øÁ¡ º¹±ÍÁß¡¦

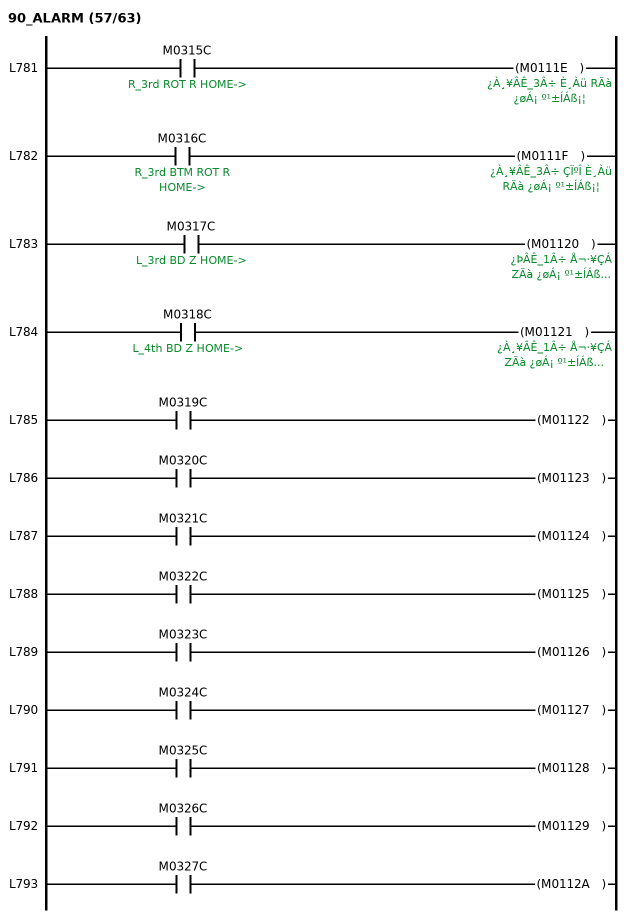
; L781
LOAD      M0315C	// R_3rd ROT R HOME->
OUT       M0111E	// ¿À¸¥ÂÊ_3Â÷ È¸Àü RÃà ¿øÁ¡ º¹±ÍÁß¡¦
; L782
LOAD      M0316C	// R_3rd BTM ROT R HOME->
OUT       M0111F	// ¿À¸¥ÂÊ_3Â÷ ÇÏºÎ È¸Àü RÃà ¿øÁ¡ º¹±ÍÁß¡¦
; L783
LOAD      M0317C	// L_3rd BD Z HOME->
OUT       M01120	// ¿ÞÂÊ_1Â÷ Å¬·¥ÇÁ ZÃà ¿øÁ¡ º¹±ÍÁß...
; L784
LOAD      M0318C	// L_4th BD Z HOME->
OUT       M01121	// ¿À¸¥ÂÊ_1Â÷ Å¬·¥ÇÁ ZÃà ¿øÁ¡ º¹±ÍÁß...
; L785
LOAD      M0319C
OUT       M01122
; L786
LOAD      M0320C
OUT       M01123
; L787
LOAD      M0321C
OUT       M01124
; L788
LOAD      M0322C
OUT       M01125
; L789
LOAD      M0323C
OUT       M01126
; L790
LOAD      M0324C
OUT       M01127
; L791
LOAD      M0325C
OUT       M01128
; L792
LOAD      M0326C
OUT       M01129
; L793
LOAD      M0327C
OUT       M0112A

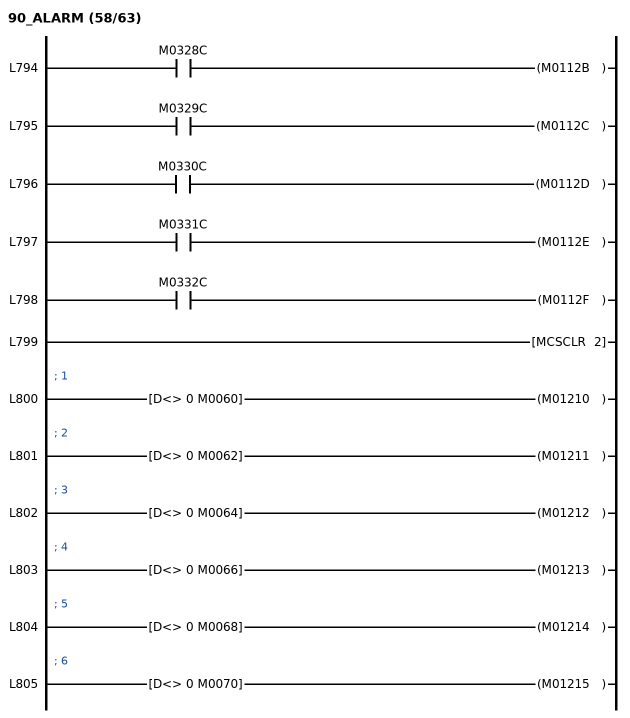
; L794
LOAD      M0328C
OUT       M0112B
; L795
LOAD      M0329C
OUT       M0112C
; L796
LOAD      M0330C
OUT       M0112D
; L797
LOAD      M0331C
OUT       M0112E
; L798
LOAD      M0332C
OUT       M0112F
; L799
MCSCLR    2
; L800
LOADD<>   0 M0060
OUT       M01210
// output comment: 1
; L801
LOADD<>   0 M0062
OUT       M01211
// output comment: 2
; L802
LOADD<>   0 M0064
OUT       M01212
// output comment: 3
; L803
LOADD<>   0 M0066
OUT       M01213
// output comment: 4
; L804
LOADD<>   0 M0068
OUT       M01214
// output comment: 5
; L805
LOADD<>   0 M0070
OUT       M01215
// output comment: 6

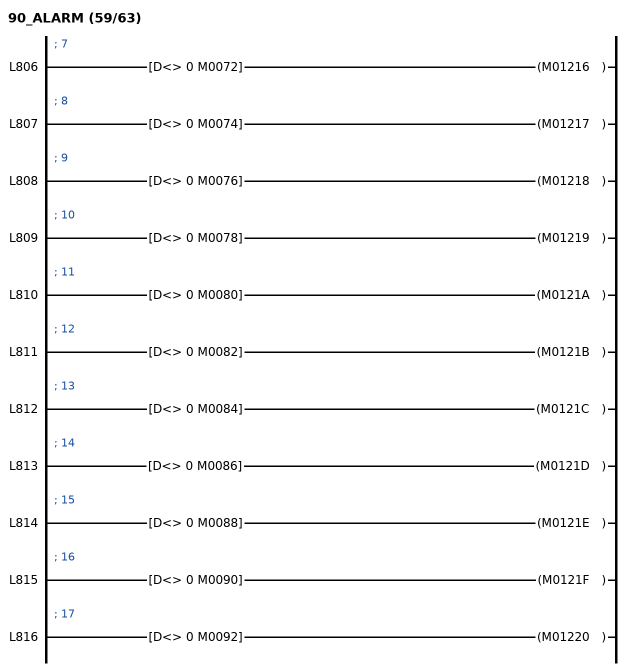
; L806
LOADD<>   0 M0072
OUT       M01216
// output comment: 7
; L807
LOADD<>   0 M0074
OUT       M01217
// output comment: 8
; L808
LOADD<>   0 M0076
OUT       M01218
// output comment: 9
; L809
LOADD<>   0 M0078
OUT       M01219
// output comment: 10
; L810
LOADD<>   0 M0080
OUT       M0121A
// output comment: 11
; L811
LOADD<>   0 M0082
OUT       M0121B
// output comment: 12
; L812
LOADD<>   0 M0084
OUT       M0121C
// output comment: 13
; L813
LOADD<>   0 M0086
OUT       M0121D
// output comment: 14
; L814
LOADD<>   0 M0088
OUT       M0121E
// output comment: 15
; L815
LOADD<>   0 M0090
OUT       M0121F
// output comment: 16
; L816
LOADD<>   0 M0092
OUT       M01220
// output comment: 17

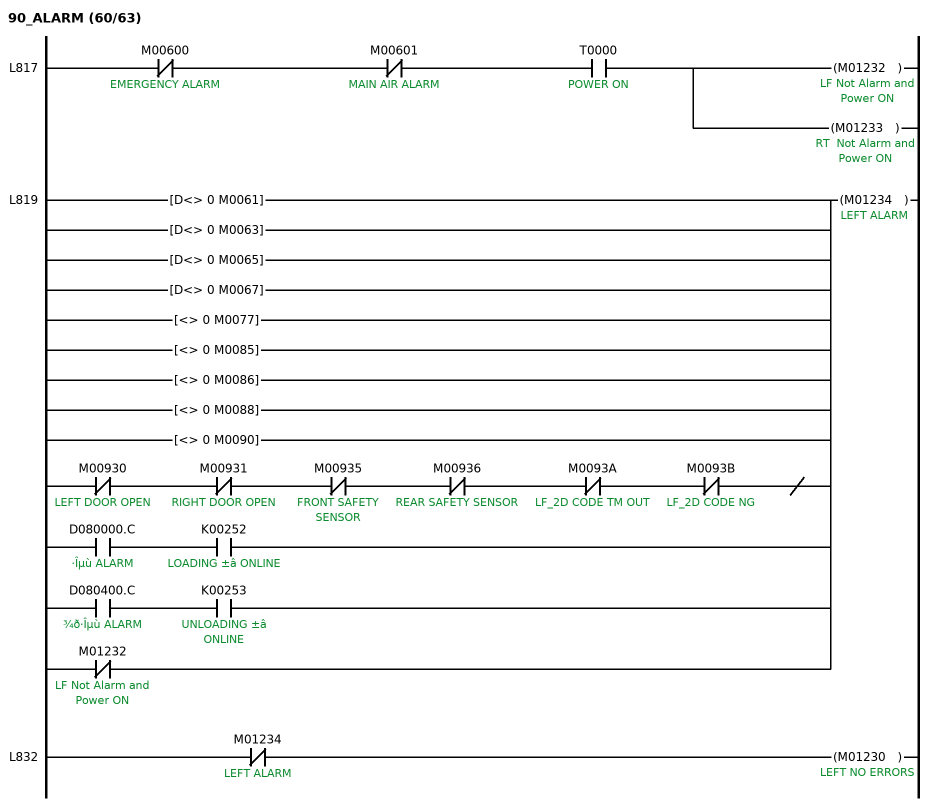
; L817
LOAD NOT  M00600	// EMERGENCY ALARM
AND NOT   M00601	// MAIN AIR ALARM
AND       T0000	// POWER ON
OUT       M01232	// LF Not Alarm and Power ON
OUT       M01233	// RT  Not Alarm and Power ON
; L819
LOADD<>   0 M0061
ORD<>     0 M0063
ORD<>     0 M0065
ORD<>     0 M0067
OR<>      0 M0077
OR<>      0 M0085
OR<>      0 M0086
OR<>      0 M0088
OR<>      0 M0090
LOAD NOT  M00930	// LEFT DOOR OPEN
AND NOT   M00931	// RIGHT DOOR OPEN
AND NOT   M00935	// FRONT SAFETY SENSOR
AND NOT   M00936	// REAR SAFETY SENSOR
AND NOT   M0093A	// LF_2D CODE TM OUT
AND NOT   M0093B	// LF_2D CODE NG
NOT
OR LOAD
LOAD      D080000.C	// ·Îµù ALARM
AND       K00252	// LOADING ±â ONLINE
OR LOAD
LOAD      D080400.C	// ¾ð·Îµù ALARM
AND       K00253	// UNLOADING ±â ONLINE
OR LOAD
OR NOT    M01232	// LF Not Alarm and Power ON
OUT       M01234	// LEFT ALARM
; L832
LOAD NOT  M01234	// LEFT ALARM
OUT       M01230	// LEFT NO ERRORS

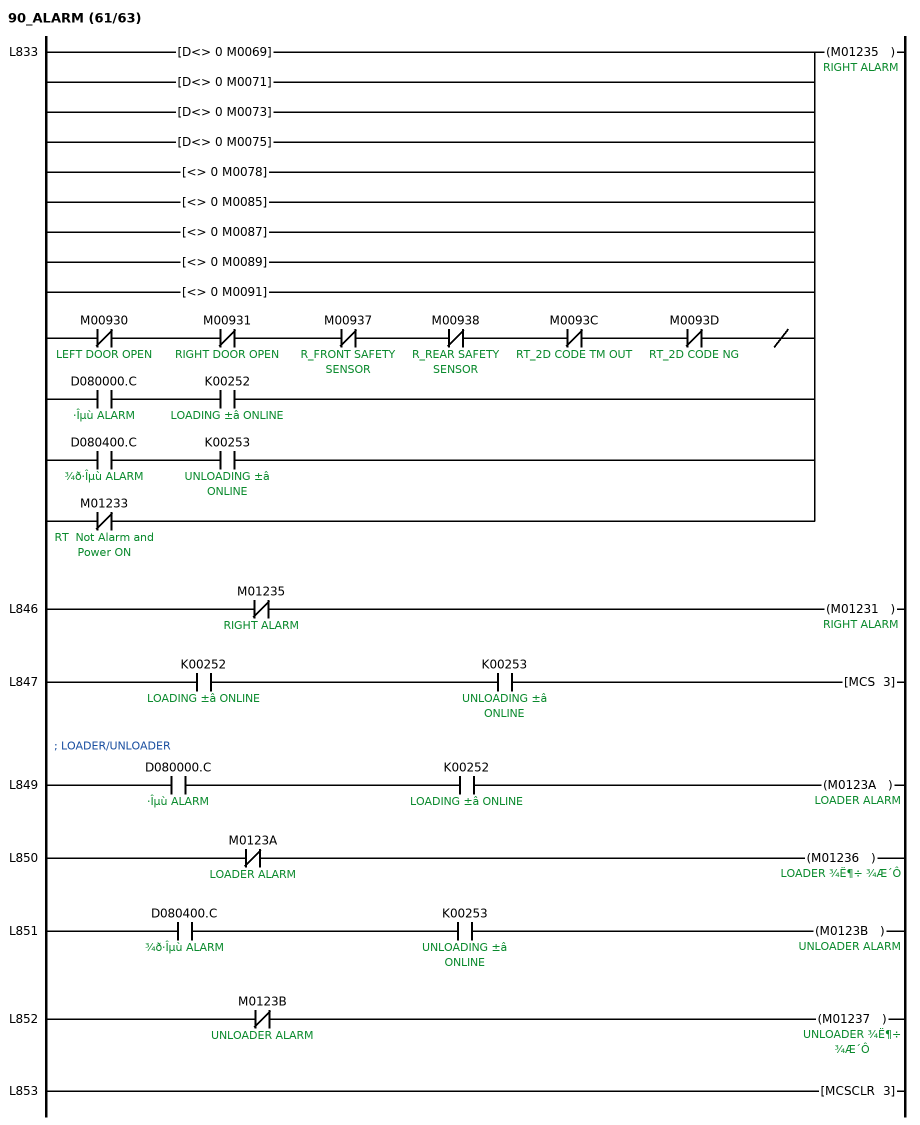
; L833
LOADD<>   0 M0069
ORD<>     0 M0071
ORD<>     0 M0073
ORD<>     0 M0075
OR<>      0 M0078
OR<>      0 M0085
OR<>      0 M0087
OR<>      0 M0089
OR<>      0 M0091
LOAD NOT  M00930	// LEFT DOOR OPEN
AND NOT   M00931	// RIGHT DOOR OPEN
AND NOT   M00937	// R_FRONT SAFETY SENSOR
AND NOT   M00938	// R_REAR SAFETY SENSOR
AND NOT   M0093C	// RT_2D CODE TM OUT
AND NOT   M0093D	// RT_2D CODE NG
NOT
OR LOAD
LOAD      D080000.C	// ·Îµù ALARM
AND       K00252	// LOADING ±â ONLINE
OR LOAD
LOAD      D080400.C	// ¾ð·Îµù ALARM
AND       K00253	// UNLOADING ±â ONLINE
OR LOAD
OR NOT    M01233	// RT  Not Alarm and Power ON
OUT       M01235	// RIGHT ALARM
; L846
LOAD NOT  M01235	// RIGHT ALARM
OUT       M01231	// RIGHT ALARM
; L847
LOAD      K00252	// LOADING ±â ONLINE
AND       K00253	// UNLOADING ±â ONLINE
MCS       3
// LOADER/UNLOADER
; L849
LOAD      D080000.C	// ·Îµù ALARM
AND       K00252	// LOADING ±â ONLINE
OUT       M0123A	// LOADER ALARM
; L850
LOAD NOT  M0123A	// LOADER ALARM
OUT       M01236	// LOADER ¾Ë¶÷ ¾Æ´Ô
; L851
LOAD      D080400.C	// ¾ð·Îµù ALARM
AND       K00253	// UNLOADING ±â ONLINE
OUT       M0123B	// UNLOADER ALARM
; L852
LOAD NOT  M0123B	// UNLOADER ALARM
OUT       M01237	// UNLOADER ¾Ë¶÷ ¾Æ´Ô
; L853
MCSCLR    3

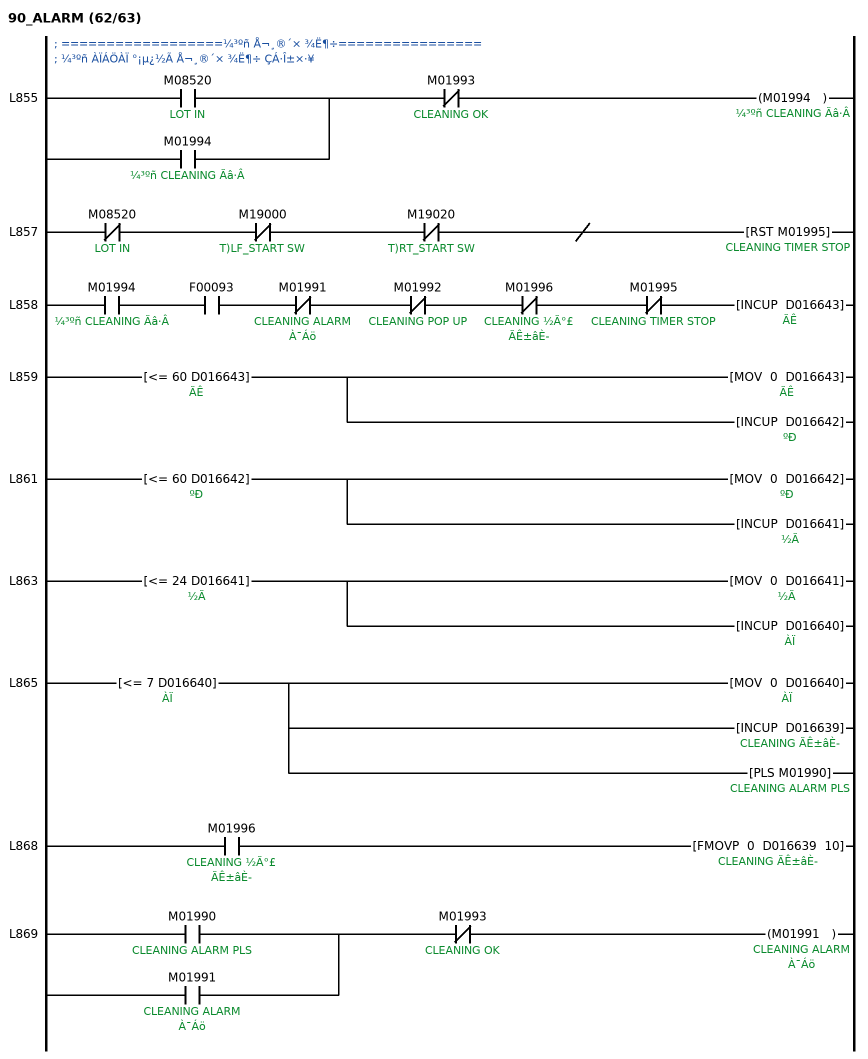
// ==================¼³ºñ Å¬¸®´× ¾Ë¶÷================
; L855
LOAD      M08520	// LOT IN
OR        M01994	// ¼³ºñ CLEANING Ãâ·Â
AND NOT   M01993	// CLEANING OK
OUT       M01994	// ¼³ºñ CLEANING Ãâ·Â
// output comment: ¼³ºñ ÀÏÁÖÀÏ °¡µ¿½Ã Å¬¸®´× ¾Ë¶÷ ÇÁ·Î±×·¥
; L857
LOAD NOT  M08520	// LOT IN
AND NOT   M19000	// T)LF_START SW
AND NOT   M19020	// T)RT_START SW
NOT
RST       M01995	// CLEANING TIMER STOP
; L858
LOAD      M01994	// ¼³ºñ CLEANING Ãâ·Â
AND       F00093
AND NOT   M01991	// CLEANING ALARM À¯Áö
AND NOT   M01992	// CLEANING POP UP
AND NOT   M01996	// CLEANING ½Ã°£ ÃÊ±âÈ­
AND NOT   M01995	// CLEANING TIMER STOP
INCUP     D016643	// ÃÊ
; L859
LOAD<=    60 D016643	// ÃÊ
MOV       0 D016643	// ÃÊ
INCUP     D016642	// ºÐ
; L861
LOAD<=    60 D016642	// ºÐ
MOV       0 D016642	// ºÐ
INCUP     D016641	// ½Ã
; L863
LOAD<=    24 D016641	// ½Ã
MOV       0 D016641	// ½Ã
INCUP     D016640	// ÀÏ
; L865
LOAD<=    7 D016640	// ÀÏ
MOV       0 D016640	// ÀÏ
INCUP     D016639	// CLEANING ÃÊ±âÈ­
OUTP      M01990	// CLEANING ALARM PLS
; L868
LOAD      M01996	// CLEANING ½Ã°£ ÃÊ±âÈ­
FMOVP     0 D016639 10	// CLEANING ÃÊ±âÈ­
; L869
LOAD      M01990	// CLEANING ALARM PLS
OR        M01991	// CLEANING ALARM À¯Áö
AND NOT   M01993	// CLEANING OK
OUT       M01991	// CLEANING ALARM À¯Áö

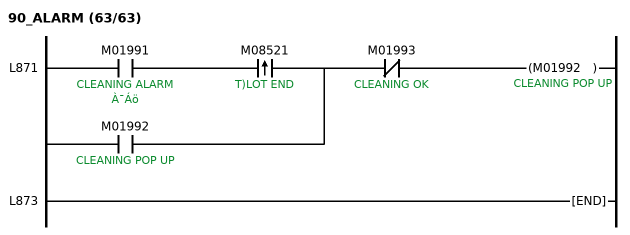
; L871
LOAD      M01991	// CLEANING ALARM À¯Áö
ANDP      M08521	// T)LOT END
OR        M01992	// CLEANING POP UP
AND NOT   M01993	// CLEANING OK
OUT       M01992	// CLEANING POP UP
; L873
END

PROGRAM 91_DEVICE_CHANGE (task: ½ºÄµ ÇÁ·Î±×·¥)

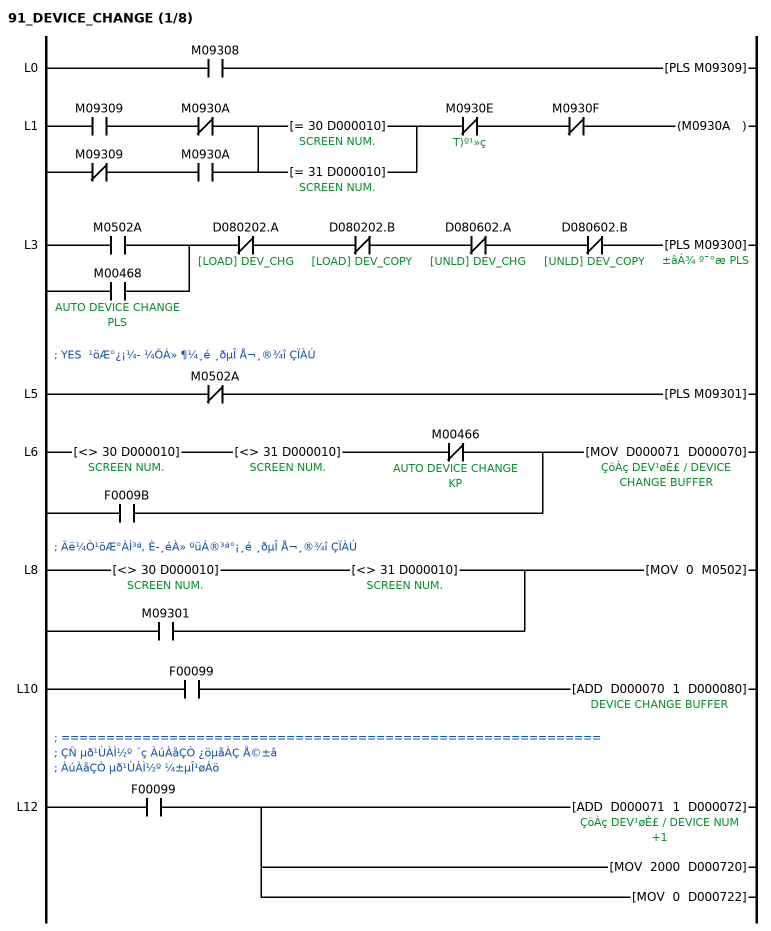
; L0
LOAD      M09308
OUTP      M09309
; L1
LOAD      M09309
AND NOT   M0930A
LOAD NOT  M09309
AND       M0930A
OR LOAD
LOAD=     30 D000010	// SCREEN NUM.
OR=       31 D000010	// SCREEN NUM.
AND LOAD
AND NOT   M0930E	// T)º¹»ç
AND NOT   M0930F
OUT       M0930A
; L3
LOAD      M0502A
OR        M00468	// AUTO DEVICE CHANGE PLS
AND NOT   D080202.A	// [LOAD] DEV_CHG
AND NOT   D080202.B	// [LOAD] DEV_COPY
AND NOT   D080602.A	// [UNLD] DEV_CHG
AND NOT   D080602.B	// [UNLD] DEV_COPY
OUTP      M09300	// ±âÁ¾ º¯°æ PLS
; L5
LOAD NOT  M0502A
OUTP      M09301
// output comment: YES  ¹öÆ°¿¡¼­ ¼ÕÀ» ¶¼¸é ¸ðµÎ Å¬¸®¾î ÇÏÀÚ
; L6
LOAD<>    30 D000010	// SCREEN NUM.
AND<>     31 D000010	// SCREEN NUM.
AND NOT   M00466	// AUTO DEVICE CHANGE KP
OR        F0009B
MOV       D000071 D000070	// ÇöÀç DEV¹øÈ£ / DEVICE CHANGE BUFFER
; L8
LOAD<>    30 D000010	// SCREEN NUM.
AND<>     31 D000010	// SCREEN NUM.
OR        M09301
MOV       0 M0502
// output comment: Ãë¼Ò¹öÆ°ÀÌ³ª, È­¸éÀ» ºüÁ®³ª°¡¸é ¸ðµÎ Å¬¸®¾î ÇÏÀÚ
; L10
LOAD      F00099
ADD       D000070 1 D000080	// DEVICE CHANGE BUFFER
// ============================================================
; L12
LOAD      F00099
ADD       D000071 1 D000072	// ÇöÀç DEV¹øÈ£ / DEVICE NUM +1
MOV       2000 D000720
MOV       0 D000722
// output comment: ÇÑ µð¹ÙÀÌ½º ´ç ÀúÀåÇÒ ¿öµåÀÇ Å©±â
// output comment: ÀúÀåÇÒ µð¹ÙÀÌ½º ¼±µÎ¹øÁö

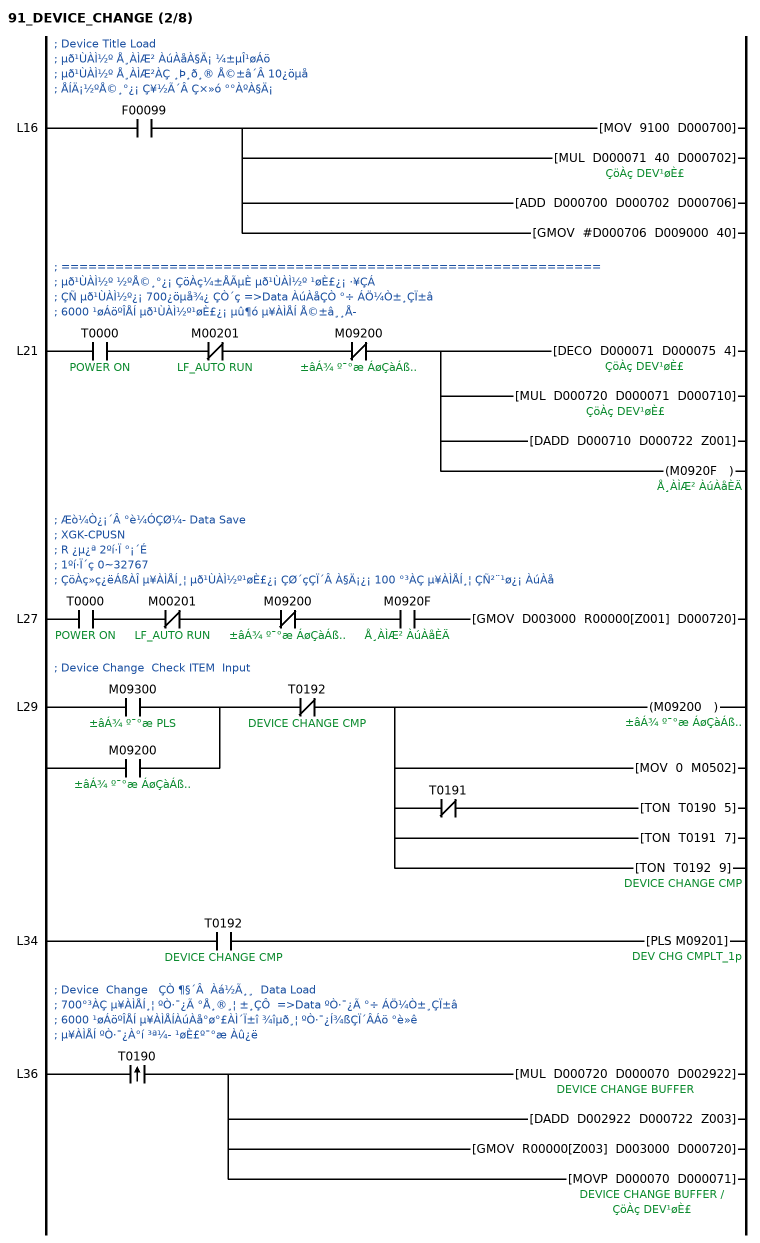
// Device Title Load
; L16
LOAD      F00099
MOV       9100 D000700
MUL       D000071 40 D000702	// ÇöÀç DEV¹øÈ£
ADD       D000700 D000702 D000706
GMOV      #D000706 D009000 40
// output comment: µð¹ÙÀÌ½º Å¸ÀÌÆ² ÀúÀåÀ§Ä¡ ¼±µÎ¹øÁö
// output comment: µð¹ÙÀÌ½º Å¸ÀÌÆ²ÀÇ ¸Þ¸ð¸® Å©±â´Â 10¿öµå
// output comment: ÅÍÄ¡½ºÅ©¸°¿¡ Ç¥½Ã´Â Ç×»ó °°ÀºÀ§Ä¡
// ============================================================
; L21
LOAD      T0000	// POWER ON
AND NOT   M00201	// LF_AUTO RUN
AND NOT   M09200	// ±âÁ¾ º¯°æ ÁøÇàÁß..
DECO      D000071 D000075 4	// ÇöÀç DEV¹øÈ£
MUL       D000720 D000071 D000710	// ÇöÀç DEV¹øÈ£
DADD      D000710 D000722 Z001
OUT       M0920F	// Å¸ÀÌÆ² ÀúÀåÈÄ
// output comment: µð¹ÙÀÌ½º ½ºÅ©¸°¿¡ ÇöÀç¼±ÅÃµÈ µð¹ÙÀÌ½º ¹øÈ£¿¡ ·¥ÇÁ
// output comment: ÇÑ µð¹ÙÀÌ½º¿¡ 700¿öµå¾¿ ÇÒ´ç =>Data ÀúÀåÇÒ °÷ ÁÖ¼Ò±¸ÇÏ±â
// output comment: 6000 ¹øÁöºÎÅÍ µð¹ÙÀÌ½º¹øÈ£¿¡ µû¶ó µ¥ÀÌÅÍ Å©±â¸¸Å­
// Æò¼Ò¿¡´Â °è¼ÓÇØ¼­ Data Save
// XGK-CPUSN
// R ¿µ¿ª 2ºí·Ï °¡´É
// 1ºí·Ï´ç 0~32767
; L27
LOAD      T0000	// POWER ON
AND NOT   M00201	// LF_AUTO RUN
AND NOT   M09200	// ±âÁ¾ º¯°æ ÁøÇàÁß..
AND       M0920F	// Å¸ÀÌÆ² ÀúÀåÈÄ
GMOV      D003000 R00000[Z001] D000720
// output comment: ÇöÀç»ç¿ëÁßÀÎ µ¥ÀÌÅÍ¸¦ µð¹ÙÀÌ½º¹øÈ£¿¡ ÇØ´çÇÏ´Â À§Ä¡¿¡ 100 °³ÀÇ µ¥ÀÌÅÍ¸¦ ÇÑ²¨¹ø¿¡ ÀúÀå
// Device Change  Check ITEM  Input
; L29
LOAD      M09300	// ±âÁ¾ º¯°æ PLS
OR        M09200	// ±âÁ¾ º¯°æ ÁøÇàÁß..
AND NOT   T0192	// DEVICE CHANGE CMP
OUT       M09200	// ±âÁ¾ º¯°æ ÁøÇàÁß..
MOV       0 M0502
MPUSH
AND NOT   T0191
TON       T0190 5
MPOP
TON       T0191 7
TON       T0192 9	// DEVICE CHANGE CMP
; L34
LOAD      T0192	// DEVICE CHANGE CMP
OUTP      M09201	// DEV CHG CMPLT_1p
// Device  Change   ÇÒ ¶§´Â  Àá½Ã¸¸  Data Load
; L36
LOADP     T0190
MUL       D000720 D000070 D002922	// DEVICE CHANGE BUFFER
DADD      D002922 D000722 Z003
GMOV      R00000[Z003] D003000 D000720
MOVP      D000070 D000071	// DEVICE CHANGE BUFFER / ÇöÀç DEV¹øÈ£
// output comment: 700°³ÀÇ µ¥ÀÌÅÍ¸¦ ºÒ·¯¿Ã °Å¸®¸¦ ±¸ÇÔ  =>Data ºÒ·¯¿Ã °÷ ÁÖ¼Ò±¸ÇÏ±â
// output comment: 6000 ¹øÁöºÎÅÍ µ¥ÀÌÅÍÀúÀå°ø°£ÀÌ´Ï±î ¾îµð¸¦ ºÒ·¯¿Í¾ßÇÏ´ÂÁö °è»ê
// output comment: µ¥ÀÌÅÍ ºÒ·¯¿À°í ³ª¼­ ¹øÈ£º¯°æ Àû¿ë

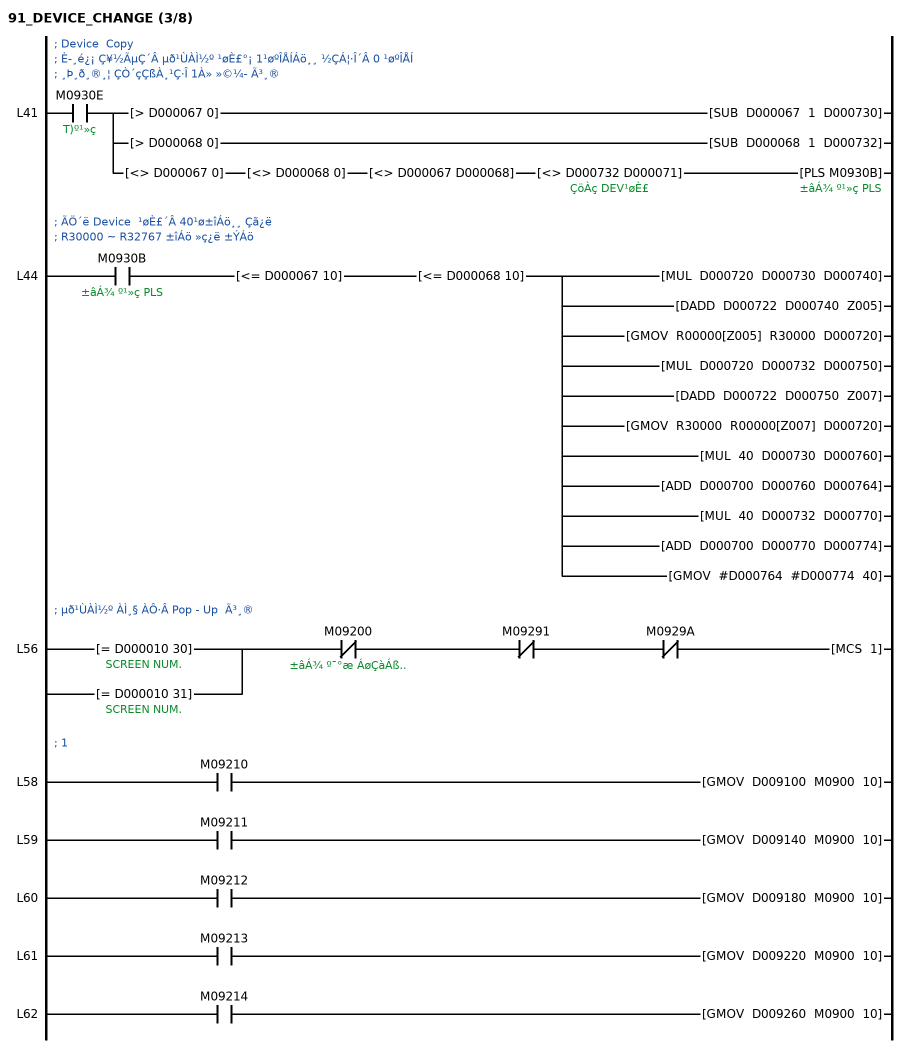
// Device  Copy
; L41
LOAD      M0930E	// T)º¹»ç
MPUSH
AND>      D000067 0
SUB       D000067 1 D000730
MLOAD
AND>      D000068 0
SUB       D000068 1 D000732
MPOP
AND<>     D000067 0
AND<>     D000068 0
AND<>     D000067 D000068
AND<>     D000732 D000071	// ÇöÀç DEV¹øÈ£
OUTP      M0930B	// ±âÁ¾ º¹»ç PLS
// output comment: È­¸é¿¡ Ç¥½ÃµÇ´Â µð¹ÙÀÌ½º ¹øÈ£°¡ 1¹øºÎÅÍÁö¸¸ ½ÇÁ¦·Î´Â 0 ¹øºÎÅÍ
// output comment: ¸Þ¸ð¸®¸¦ ÇÒ´çÇßÀ¸¹Ç·Î 1À» »©¼­ Ã³¸®
; L44
LOAD      M0930B	// ±âÁ¾ º¹»ç PLS
AND<=     D000067 10
AND<=     D000068 10
MUL       D000720 D000730 D000740
DADD      D000722 D000740 Z005
GMOV      R00000[Z005] R30000 D000720
MUL       D000720 D000732 D000750
DADD      D000722 D000750 Z007
GMOV      R30000 R00000[Z007] D000720
MUL       40 D000730 D000760
ADD       D000700 D000760 D000764
MUL       40 D000732 D000770
ADD       D000700 D000770 D000774
GMOV      #D000764 #D000774 40
// output comment: ÃÖ´ë Device  ¹øÈ£´Â 40¹ø±îÁö¸¸ Çã¿ë
// output comment: R30000 ~ R32767 ±îÁö »ç¿ë ±ÝÁö
// µð¹ÙÀÌ½º ÀÌ¸§ ÀÔ·Â Pop - Up  Ã³¸®
; L56
LOAD=     D000010 30	// SCREEN NUM.
OR=       D000010 31	// SCREEN NUM.
AND NOT   M09200	// ±âÁ¾ º¯°æ ÁøÇàÁß..
AND NOT   M09291
AND NOT   M0929A
MCS       1
; L58
LOAD      M09210
GMOV      D009100 M0900 10
// output comment: 1
; L59
LOAD      M09211
GMOV      D009140 M0900 10
; L60
LOAD      M09212
GMOV      D009180 M0900 10
; L61
LOAD      M09213
GMOV      D009220 M0900 10
; L62
LOAD      M09214
GMOV      D009260 M0900 10

